KUKA KRL program: MyProgram_079().src

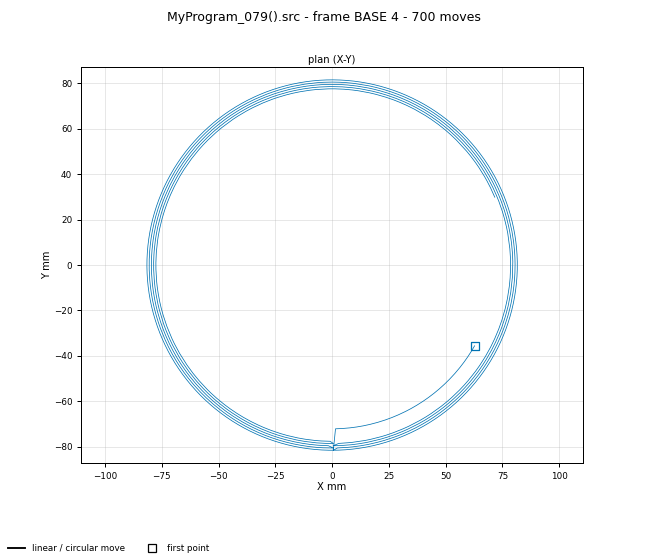
[picture p0: tool path of MyProgram_079().src in frame BASE 4, 700 of 700 moves have a stored position in this frame; points joined in program order, loops and branches not executed]
&ACCESS RVP
&REL 1
&PARAM TEMPLATE = C:\KRC\Roboter\Template\vorgabe
&PARAM EDITMASK = *
DEF MyProgram_079()
; ---- Setting reference (Base) ----
$BASE = BASE_DATA[4]

; --------------------------
; ---- Setting tool (TCP) ----
$TOOL = TOOL_DATA[3]
; --------------------------

$VEL.CP = VEL_APROX_PRINT
Startdeposition()
$VEL.CP = VEL_PRINT
LIN {X 62.743,Y -35.5612,Z 80,A -35.5056,B 24.9021,C -2.2844,E1 25.1384,E2 119.903} C_DIS
LIN {X 61.3969,Y -37.8376,Z 80,A -37.6345,B 24.9027,C -2.2777,E1 25.1353,E2 122.037} C_DIS
LIN {X 59.7597,Y -40.3719,Z 80,A -39.9948,B 24.9032,C -2.2721,E1 25.1316,E2 124.3987} C_DIS
LIN {X 58.1912,Y -42.6015,Z 80,A -42.2134,B 24.9038,C -2.2647,E1 25.128,E2 126.624} C_DIS
LIN {X 56.2909,Y -45.0843,Z 80,A -44.7326,B 24.9044,C -2.2572,E1 25.1237,E2 129.1493} C_DIS
LIN {X 54.0306,Y -47.7691,Z 80,A -47.4805,B 24.9049,C -2.2512,E1 25.1187,E2 131.8988} C_DIS
LIN {X 51.744,Y -50.2367,Z 80,A -50.1078,B 24.9054,C -2.2459,E1 25.1136,E2 134.5273} C_DIS
LIN {X 49.5214,Y -52.4286,Z 80,A -52.5294,B 24.9057,C -2.2416,E1 25.1087,E2 136.9488} C_DIS
LIN {X 47.2452,Y -54.4891,Z 80,A -54.9859,B 24.9062,C -2.2356,E1 25.1036,E2 139.4099} C_DIS
LIN {X 44.8927,Y -56.4428,Z 80,A -57.3886,B 24.9066,C -2.231,E1 25.0984,E2 141.8143} C_DIS
LIN {X 42.5333,Y -58.2412,Z 80,A -59.7773,B 24.9071,C -2.2252,E1 25.093,E2 144.2081} C_DIS
LIN {X 40.0623,Y -59.9686,Z 80,A -62.2006,B 24.9076,C -2.2197,E1 25.0874,E2 146.6363} C_DIS
LIN {X 37.263,Y -61.7465,Z 80,A -64.7758,B 24.9079,C -2.2164,E1 25.0813,E2 149.2111} C_DIS
LIN {X 34.7417,Y -63.2004,Z 80,A -67.0445,B 24.9081,C -2.2135,E1 25.0758,E2 151.4799} C_DIS
LIN {X 32.4215,Y -64.4207,Z 80,A -69.2156,B 24.9086,C -2.2077,E1 25.0704,E2 153.6588} C_DIS
LIN {X 29.2273,Y -65.9316,Z 80,A -72.0556,B 24.909,C -2.2025,E1 25.0632,E2 156.504} C_DIS
LIN {X 26.2757,Y -67.1618,Z 80,A -74.4953,B 24.909,C -2.2017,E1 25.0569,E2 158.9402} C_DIS
LIN {X 23.4466,Y -68.2022,Z 80,A -76.9337,B 24.9094,C -2.1974,E1 25.0504,E2 161.3837} C_DIS
LIN {X 20.0842,Y -69.2668,Z 80,A -79.7346,B 24.9097,C -2.1942,E1 25.0429,E2 164.1871} C_DIS
LIN {X 16.6714,Y -70.165,Z 80,A -82.321,B 24.9094,C -2.1972,E1 25.036,E2 166.7625} C_DIS
LIN {X 13.7247,Y -70.8008,Z 80,A -84.7485,B 24.9097,C -2.1943,E1 25.0293,E2 169.194} C_DIS
LIN {X 10.8752,Y -71.2942,Z 80,A -87.1416,B 24.91,C -2.1901,E1 25.0227,E2 171.5947} C_DIS
LIN {X 7.9418,Y -71.6799,Z 80,A -89.5264,B 24.9102,C -2.1877,E1 25.0161,E2 173.9832} C_DIS
LIN {X 4.4201,Y -71.9832,Z 80,A -92.175,B 24.91,C -2.1906,E1 25.0087,E2 176.6238} C_DIS
LIN {X 1.499,Y -72.1033,Z 80,A -94.5519,B 24.9102,C -2.1884,E1 25.0021,E2 179.0053} C_DIS
LIN {X 1.499,Y -72.1033,Z 80,A -94.5519,B 24.9102,C -2.1884,E1 25.0021,E2 179.0053} C_DIS
Enddeposition()
LIN {X 0.5368,Y -81.5501,Z 81,A -94.2827,B 24.9204,C -2.0597,E1 25.002,E2 179.0416} C_DIS
Startdeposition()
$VEL.CP = VEL_PRINT
LIN {X -1.5341,Y -81.5397,Z 81,A -96.3673,B 24.9219,C -2.0407,E1 24.996,E2 181.1713} C_DIS
LIN {X -4.4685,Y -81.4316,Z 81,A -98.4471,B 24.9219,C -2.04,E1 24.9902,E2 183.2532} C_DIS
LIN {X -7.4627,Y -81.212,Z 81,A -100.5636,B 24.9219,C -2.0399,E1 24.9843,E2 185.371} C_DIS
LIN {X -10.4468,Y -80.8822,Z 81,A -102.6737,B 24.9219,C -2.0401,E1 24.9785,E2 187.4818} C_DIS
LIN {X -13.4168,Y -80.4429,Z 81,A -104.7842,B 24.9219,C -2.0407,E1 24.9727,E2 189.593} C_DIS
LIN {X -16.4332,Y -79.8813,Z 81,A -106.9178,B 24.9219,C -2.0421,E1 24.9668,E2 191.7254} C_DIS
LIN {X -19.3623,Y -79.2223,Z 81,A -109.0295,B 24.9217,C -2.0431,E1 24.9611,E2 193.8376} C_DIS
LIN {X -22.2651,Y -78.456,Z 81,A -111.1414,B 24.9217,C -2.0443,E1 24.9554,E2 195.9499} C_DIS
LIN {X -25.075,Y -77.6036,Z 81,A -113.2323,B 24.9216,C -2.045,E1 24.9498,E2 198.0427} C_DIS
LIN {X -27.9764,Y -76.6055,Z 81,A -115.3677,B 24.9214,C -2.0474,E1 24.9442,E2 200.1766} C_DIS
LIN {X -30.716,Y -75.5487,Z 81,A -117.4594,B 24.9214,C -2.0486,E1 24.9387,E2 202.27} C_DIS
LIN {X -33.4759,Y -74.3669,Z 81,A -119.5737,B 24.9211,C -2.0507,E1 24.9333,E2 204.3844} C_DIS
LIN {X -36.1904,Y -73.0844,Z 81,A -121.6887,B 24.921,C -2.053,E1 24.928,E2 206.4993} C_DIS
LIN {X -38.9139,Y -71.6713,Z 81,A -123.8262,B 24.9207,C -2.0563,E1 24.9227,E2 208.6349} C_DIS
LIN {X -41.4688,Y -70.224,Z 81,A -125.9198,B 24.9206,C -2.0583,E1 24.9177,E2 210.73} C_DIS
LIN {X -44.0254,Y -68.6501,Z 81,A -128.0364,B 24.9203,C -2.0613,E1 24.9127,E2 212.8462} C_DIS
LIN {X -46.5224,Y -66.9831,Z 81,A -130.1279,B 24.92,C -2.0652,E1 24.9078,E2 214.9355} C_DIS
LIN {X -48.9564,Y -65.2254,Z 81,A -132.2705,B 24.9198,C -2.0679,E1 24.903,E2 217.0793} C_DIS
LIN {X -51.3752,Y -63.3377,Z 81,A -134.4108,B 24.9195,C -2.0722,E1 24.8983,E2 219.2173} C_DIS
LIN {X -53.5934,Y -61.4722,Z 81,A -136.4946,B 24.9193,C -2.0747,E1 24.8939,E2 221.303} C_DIS
LIN {X -55.8954,Y -59.3867,Z 81,A -138.6479,B 24.9189,C -2.0799,E1 24.8895,E2 223.4528} C_DIS
LIN {X -58.0434,Y -57.2891,Z 81,A -140.7613,B 24.9185,C -2.0841,E1 24.8853,E2 225.5649} C_DIS
LIN {X -60.0681,Y -55.1624,Z 81,A -142.8642,B 24.9183,C -2.0875,E1 24.8813,E2 227.6689} C_DIS
LIN {X -62.1006,Y -52.8639,Z 81,A -145.0065,B 24.9179,C -2.0928,E1 24.8774,E2 229.8084} C_DIS
LIN {X -64.0043,Y -50.5423,Z 81,A -147.127,B 24.9175,C -2.0974,E1 24.8736,E2 231.9278} C_DIS
LIN {X -65.8212,Y -48.1523,Z 81,A -149.2477,B 24.9171,C -2.1022,E1 24.8701,E2 234.0473} C_DIS
LIN {X -67.512,Y -45.7516,Z 81,A -151.3463,B 24.9168,C -2.1064,E1 24.8668,E2 236.1462} C_DIS
LIN {X -69.1852,Y -43.1797,Z 81,A -153.4902,B 24.9163,C -2.1122,E1 24.8635,E2 238.287} C_DIS
LIN {X -70.6947,Y -40.6611,Z 81,A -155.5896,B 24.916,C -2.1167,E1 24.8606,E2 240.3866} C_DIS
LIN {X -72.1435,Y -38.0315,Z 81,A -157.7117,B 24.9155,C -2.122,E1 24.8577,E2 242.5072} C_DIS
LIN {X -73.523,Y -35.2909,Z 81,A -159.8565,B 24.915,C -2.1283,E1 24.8551,E2 244.6487} C_DIS
LIN {X -74.7458,Y -32.6212,Z 81,A -161.9566,B 24.9147,C -2.1331,E1 24.8527,E2 246.7488} C_DIS
LIN {X -75.8703,Y -29.9127,Z 81,A -164.0576,B 24.9143,C -2.1379,E1 24.8505,E2 248.85} C_DIS
LIN {X -76.9648,Y -26.972,Z 81,A -166.2057,B 24.9136,C -2.1458,E1 24.8485,E2 250.9914} C_DIS
LIN {X -77.8859,Y -24.1838,Z 81,A -168.3262,B 24.9133,C -2.1505,E1 24.8466,E2 253.113} C_DIS
LIN {X -78.7405,Y -21.237,Z 81,A -170.4721,B 24.9127,C -2.1572,E1 24.845,E2 255.2552} C_DIS
LIN {X -79.4688,Y -18.3244,Z 81,A -172.5959,B 24.9122,C -2.1632,E1 24.8436,E2 257.377} C_DIS
LIN {X -80.0894,Y -15.3869,Z 81,A -174.7195,B 24.9117,C -2.1693,E1 24.8424,E2 259.4986} C_DIS
LIN {X -80.6015,Y -12.4286,Z 81,A -176.8435,B 24.9112,C -2.1755,E1 24.8415,E2 261.6205} C_DIS
LIN {X -80.9967,Y -9.519,Z 81,A -178.9453,B 24.9108,C -2.181,E1 24.8407,E2 263.7219} C_DIS
LIN {X -81.2974,Y -6.4656,Z 81,A 178.9082,B 24.9102,C -2.188,E1 24.8402,E2 265.8645} C_DIS
LIN {X -81.4775,Y -3.5347,Z 81,A 176.806,B 24.9097,C -2.1935,E1 24.8399,E2 267.9661} C_DIS
LIN {X -81.553,Y -0.483,Z 81,A 174.6524,B 24.9092,C -2.2001,E1 24.8398,E2 270.117} C_DIS
LIN {X -81.5167,Y 2.4687,Z 81,A 172.5572,B 24.9087,C -2.2062,E1 24.8399,E2 272.2103} C_DIS
LIN {X -81.3662,Y 5.5332,Z 81,A 170.4187,B 24.9081,C -2.2135,E1 24.8402,E2 274.3443} C_DIS
LIN {X -81.1074,Y 8.5243,Z 81,A 168.2859,B 24.9076,C -2.2196,E1 24.8408,E2 276.4752} C_DIS
LIN {X -80.7479,Y 11.4386,Z 81,A 166.1841,B 24.9071,C -2.2252,E1 24.8416,E2 278.5763} C_DIS
LIN {X -80.2605,Y 14.4679,Z 81,A 164.0373,B 24.9065,C -2.2322,E1 24.8426,E2 280.7189} C_DIS
LIN {X -79.6736,Y 17.4122,Z 81,A 161.9133,B 24.906,C -2.2385,E1 24.8438,E2 282.8406} C_DIS
LIN {X -78.9787,Y 20.333,Z 81,A 159.7888,B 24.9055,C -2.2447,E1 24.8452,E2 284.9625} C_DIS
LIN {X -78.1956,Y 23.163,Z 81,A 157.6873,B 24.905,C -2.2502,E1 24.8468,E2 287.0633} C_DIS
LIN {X -77.29,Y 26.0255,Z 81,A 155.5633,B 24.9045,C -2.2563,E1 24.8486,E2 289.1848} C_DIS
LIN {X -76.2564,Y 28.9143,Z 81,A 153.4169,B 24.9039,C -2.2631,E1 24.8507,E2 291.3269} C_DIS
LIN {X -75.1404,Y 31.7015,Z 81,A 151.2934,B 24.9034,C -2.2691,E1 24.8529,E2 293.448} C_DIS
LIN {X -73.9505,Y 34.386,Z 81,A 149.1924,B 24.903,C -2.2743,E1 24.8553,E2 295.5481} C_DIS
LIN {X -72.6348,Y 37.0846,Z 81,A 147.0693,B 24.9025,C -2.2801,E1 24.858,E2 297.6687} C_DIS
LIN {X -71.2206,Y 39.7329,Z 81,A 144.9462,B 24.902,C -2.2859,E1 24.8608,E2 299.7893} C_DIS
LIN {X -69.6756,Y 42.3838,Z 81,A 142.801,B 24.9014,C -2.2923,E1 24.8639,E2 301.9304} C_DIS
LIN {X -68.1046,Y 44.8646,Z 81,A 140.7009,B 24.901,C -2.297,E1 24.867,E2 304.0297} C_DIS
LIN {X -66.3689,Y 47.3946,Z 81,A 138.5564,B 24.9005,C -2.3032,E1 24.8705,E2 306.1701} C_DIS
LIN {X -64.6197,Y 49.7531,Z 81,A 136.4568,B 24.9001,C -2.3077,E1 24.874,E2 308.2689} C_DIS
LIN {X -62.8228,Y 52.0037,Z 81,A 134.3726,B 24.8998,C -2.3114,E1 24.8777,E2 310.3541} C_DIS
LIN {X -60.7405,Y 54.4211,Z 81,A 132.1915,B 24.8991,C -2.3186,E1 24.8817,E2 312.5278} C_DIS
LIN {X -58.6963,Y 56.62,Z 81,A 130.0707,B 24.8987,C -2.3235,E1 24.8857,E2 314.6462} C_DIS
LIN {X -56.5725,Y 58.742,Z 81,A 127.9501,B 24.8983,C -2.3282,E1 24.8899,E2 316.7645} C_DIS
LIN {X -54.372,Y 60.7845,Z 81,A 125.8299,B 24.8979,C -2.3327,E1 24.8943,E2 318.8824} C_DIS
LIN {X -52.1486,Y 62.7025,Z 81,A 123.7326,B 24.8976,C -2.3364,E1 24.8988,E2 320.9791} C_DIS
LIN {X -49.8053,Y 64.5794,Z 81,A 121.6131,B 24.8972,C -2.3406,E1 24.9034,E2 323.0965} C_DIS
LIN {X -47.3409,Y 66.4072,Z 81,A 119.4718,B 24.8968,C -2.3453,E1 24.9082,E2 325.2339} C_DIS
LIN {X -44.8646,Y 68.1046,Z 81,A 117.3614,B 24.8964,C -2.3494,E1 24.9131,E2 327.3417} C_DIS
LIN {X -42.3838,Y 69.6756,Z 81,A 115.2575,B 24.8962,C -2.3521,E1 24.9181,E2 329.4458} C_DIS
LIN {X -39.7905,Y 71.1884,Z 81,A 113.1399,B 24.8959,C -2.3556,E1 24.9232,E2 331.5613} C_DIS
LIN {X -37.0846,Y 72.6348,Z 81,A 111.0093,B 24.8955,C -2.3598,E1 24.9285,E2 333.6877} C_DIS
LIN {X -34.386,Y 73.9505,Z 81,A 108.8838,B 24.8953,C -2.3626,E1 24.9338,E2 335.8119} C_DIS
LIN {X -31.7015,Y 75.1404,Z 81,A 106.7899,B 24.8951,C -2.3648,E1 24.9392,E2 337.9057} C_DIS
LIN {X -28.8526,Y 76.2797,Z 81,A 104.652,B 24.8948,C -2.3682,E1 24.9447,E2 340.0401} C_DIS
LIN {X -26.0255,Y 77.29,Z 81,A 102.5368,B 24.8945,C -2.3706,E1 24.9503,E2 342.1536} C_DIS
LIN {X -23.163,Y 78.1956,Z 81,A 100.4222,B 24.8943,C -2.3728,E1 24.956,E2 344.2666} C_DIS
LIN {X -20.333,Y 78.9787,Z 81,A 98.3306,B 24.8943,C -2.3741,E1 24.9616,E2 346.3584} C_DIS
LIN {X -17.4122,Y 79.6736,Z 81,A 96.2169,B 24.8941,C -2.3759,E1 24.9673,E2 348.4706} C_DIS
LIN {X -14.4679,Y 80.2605,Z 81,A 94.1037,B 24.8939,C -2.3774,E1 24.9731,E2 350.5824} C_DIS
LIN {X -11.4386,Y 80.7479,Z 81,A 91.9688,B 24.8938,C -2.3795,E1 24.979,E2 352.7143} C_DIS
LIN {X -8.5243,Y 81.1074,Z 81,A 89.8792,B 24.8938,C -2.3799,E1 24.9848,E2 354.8043} C_DIS
LIN {X -5.5332,Y 81.3662,Z 81,A 87.7676,B 24.8936,C -2.3807,E1 24.9907,E2 356.9147} C_DIS
LIN {X -2.4687,Y 81.5167,Z 81,A 85.6344,B 24.8936,C -2.3821,E1 24.9966,E2 359.0452} C_DIS
LIN {X 0.4674,Y 81.5528,Z 81,A 83.5466,B 24.8936,C -2.3818,E1 25.0025,E2 361.1337} C_DIS
LIN {X 3.5347,Y 81.4775,Z 81,A 81.4145,B 24.8935,C -2.3827,E1 25.0084,E2 363.2631} C_DIS
LIN {X 6.4656,Y 81.2974,Z 81,A 79.3276,B 24.8935,C -2.3819,E1 25.0142,E2 365.3509} C_DIS
LIN {X 9.519,Y 80.9967,Z 81,A 77.1965,B 24.8935,C -2.3823,E1 25.0201,E2 367.4796} C_DIS
LIN {X 12.4938,Y 80.5914,Z 81,A 75.0884,B 24.8935,C -2.3818,E1 25.026,E2 369.5871} C_DIS
LIN {X 15.3869,Y 80.0894,Z 81,A 73.0029,B 24.8937,C -2.3804,E1 25.0317,E2 371.6737} C_DIS
LIN {X 18.3244,Y 79.4688,Z 81,A 70.896,B 24.8937,C -2.3794,E1 25.0374,E2 373.7801} C_DIS
LIN {X 21.237,Y 78.7405,Z 81,A 68.7893,B 24.8939,C -2.3782,E1 25.0431,E2 375.8864} C_DIS
LIN {X 24.1838,Y 77.8859,Z 81,A 66.661,B 24.8939,C -2.3774,E1 25.0488,E2 378.0127} C_DIS
LIN {X 26.972,Y 76.9648,Z 81,A 64.5779,B 24.8941,C -2.3751,E1 25.0543,E2 380.0972} C_DIS
LIN {X 29.8479,Y 75.8958,Z 81,A 62.4507,B 24.8943,C -2.3739,E1 25.0599,E2 382.2227} C_DIS
LIN {X 32.6212,Y 74.7458,Z 81,A 60.347,B 24.8944,C -2.3718,E1 25.0653,E2 384.3264} C_DIS
LIN {X 35.3503,Y 73.4944,Z 81,A 58.2425,B 24.8946,C -2.3695,E1 25.0706,E2 386.431} C_DIS
LIN {X 38.0315,Y 72.1435,Z 81,A 56.139,B 24.8949,C -2.367,E1 25.0758,E2 388.5346} C_DIS
LIN {X 40.6611,Y 70.6947,Z 81,A 54.0363,B 24.8951,C -2.3643,E1 25.081,E2 390.6376} C_DIS
LIN {X 43.1797,Y 69.1852,Z 81,A 51.9561,B 24.8954,C -2.3607,E1 25.0859,E2 392.7198} C_DIS
LIN {X 45.7516,Y 67.512,Z 81,A 49.8319,B 24.8956,C -2.3582,E1 25.0909,E2 394.8428} C_DIS
LIN {X 48.2055,Y 65.7822,Z 81,A 47.7307,B 24.8959,C -2.3549,E1 25.0956,E2 396.9445} C_DIS
LIN {X 50.5941,Y 63.9634,Z 81,A 45.6295,B 24.8963,C -2.3514,E1 25.1003,E2 399.0464} C_DIS
LIN {X 52.8639,Y 62.1006,Z 81,A 43.551,B 24.8966,C -2.347,E1 25.1047,E2 401.1272} C_DIS
LIN {X 55.1138,Y 60.1127,Z 81,A 41.4509,B 24.897,C -2.3431,E1 25.1091,E2 403.2281} C_DIS
LIN {X 57.2891,Y 58.0434,Z 81,A 39.3512,B 24.8973,C -2.339,E1 25.1133,E2 405.3287} C_DIS
LIN {X 59.3867,Y 55.8954,Z 81,A 37.2519,B 24.8977,C -2.3348,E1 25.1174,E2 407.4289} C_DIS
LIN {X 61.4472,Y 53.622,Z 81,A 35.1661,B 24.898,C -2.3321,E1 25.1213,E2 409.5117} C_DIS
LIN {X 63.3377,Y 51.3752,Z 81,A 33.0545,B 24.8985,C -2.3258,E1 25.125,E2 411.6285} C_DIS
LIN {X 65.1857,Y 49.0091,Z 81,A 30.9562,B 24.8989,C -2.3211,E1 25.1286,E2 413.728} C_DIS
LIN {X 66.9585,Y 46.5578,Z 81,A 28.8509,B 24.8993,C -2.3165,E1 25.132,E2 415.8341} C_DIS
LIN {X 68.6144,Y 44.081,Z 81,A 26.7609,B 24.8998,C -2.3112,E1 25.1352,E2 417.926} C_DIS
LIN {X 70.1905,Y 41.5256,Z 81,A 24.6638,B 24.9002,C -2.3061,E1 25.1383,E2 420.0245} C_DIS
LIN {X 71.7028,Y 38.8559,Z 81,A 22.5447,B 24.9006,C -2.3015,E1 25.1411,E2 422.1435} C_DIS
LIN {X 73.0551,Y 36.2495,Z 81,A 20.4705,B 24.9011,C -2.2954,E1 25.1438,E2 424.221} C_DIS
LIN {X 74.3398,Y 33.536,Z 81,A 18.374,B 24.9016,C -2.2899,E1 25.1462,E2 426.3191} C_DIS
LIN {X 75.5487,Y 30.716,Z 81,A 16.2558,B 24.902,C -2.285,E1 25.1485,E2 428.4373} C_DIS
LIN {X 76.6281,Y 27.9144,Z 81,A 14.16,B 24.9025,C -2.2793,E1 25.1506,E2 430.535} C_DIS
LIN {X 77.5833,Y 25.1378,Z 81,A 12.0866,B 24.9031,C -2.2728,E1 25.1524,E2 432.6119} C_DIS
LIN {X 78.456,Y 22.2651,Z 81,A 9.9911,B 24.9036,C -2.2669,E1 25.1541,E2 434.7093} C_DIS
LIN {X 79.2379,Y 19.2982,Z 81,A 7.8736,B 24.904,C -2.2616,E1 25.1555,E2 436.8272} C_DIS
LIN {X 79.8813,Y 16.4332,Z 81,A 5.8008,B 24.9046,C -2.255,E1 25.1568,E2 438.9036} C_DIS
LIN {X 80.4429,Y 13.4168,Z 81,A 3.6837,B 24.9051,C -2.2495,E1 25.1578,E2 441.0211} C_DIS
LIN {X 80.8822,Y 10.4468,Z 81,A 1.5889,B 24.9056,C -2.2434,E1 25.1586,E2 443.1181} C_DIS
LIN {X 81.212,Y 7.4627,Z 81,A -0.506,B 24.9061,C -2.2372,E1 25.1592,E2 445.2151} C_DIS
LIN {X 81.4316,Y 4.4685,Z 81,A -2.6004,B 24.9066,C -2.231,E1 25.1596,E2 447.3118} C_DIS
LIN {X 81.5397,Y 1.5341,Z 81,A -4.6754,B 24.9072,C -2.2241,E1 25.1598,E2 449.3908} C_DIS
LIN {X 81.5311,Y -2.0015,Z 81,A -7.2342,B 24.9081,C -2.2137,E1 25.1597,E2 451.9589} C_DIS
LIN {X 81.4022,Y -5.0011,Z 81,A -9.321,B 24.9086,C -2.2077,E1 25.1594,E2 454.0475} C_DIS
LIN {X 81.1736,Y -7.8785,Z 81,A -11.3675,B 24.9092,C -2.2006,E1 25.1589,E2 456.0985} C_DIS
LIN {X 80.8137,Y -10.9758,Z 81,A -13.51,B 24.9096,C -2.1952,E1 25.1581,E2 458.2412} C_DIS
LIN {X 80.355,Y -13.9429,Z 81,A -15.6046,B 24.9101,C -2.1889,E1 25.1572,E2 460.3382} C_DIS
LIN {X 79.7873,Y -16.8911,Z 81,A -17.699,B 24.9106,C -2.1827,E1 25.156,E2 462.435} C_DIS
LIN {X 79.1115,Y -19.8164,Z 81,A -19.7938,B 24.9111,C -2.1766,E1 25.1546,E2 464.5323} C_DIS
LIN {X 78.3285,Y -22.7149,Z 81,A -21.9076,B 24.9117,C -2.1698,E1 25.153,E2 466.6499} C_DIS
LIN {X 77.4394,Y -25.5825,Z 81,A -23.9836,B 24.9121,C -2.1643,E1 25.1513,E2 468.7271} C_DIS
LIN {X 76.4453,Y -28.4155,Z 81,A -26.0978,B 24.9127,C -2.1577,E1 25.1492,E2 470.8451} C_DIS
LIN {X 75.3476,Y -31.21,Z 81,A -28.1931,B 24.9132,C -2.1517,E1 25.1471,E2 472.9429} C_DIS
LIN {X 74.1478,Y -33.9622,Z 81,A -30.2692,B 24.9136,C -2.1465,E1 25.1447,E2 475.0202} C_DIS
LIN {X 72.8475,Y -36.6683,Z 81,A -32.384,B 24.9141,C -2.1401,E1 25.1421,E2 477.1388} C_DIS
LIN {X 71.4485,Y -39.3248,Z 81,A -34.4799,B 24.9146,C -2.1343,E1 25.1393,E2 479.2371} C_DIS
LIN {X 69.9526,Y -41.928,Z 81,A -36.5568,B 24.915,C -2.1293,E1 25.1363,E2 481.3152} C_DIS
LIN {X 68.362,Y -44.4743,Z 81,A -38.6723,B 24.9155,C -2.1232,E1 25.1332,E2 483.4345} C_DIS
LIN {X 66.6787,Y -46.9604,Z 81,A -40.7495,B 24.9158,C -2.1184,E1 25.1299,E2 485.5128} C_DIS
LIN {X 64.905,Y -49.3828,Z 81,A -42.8464,B 24.9163,C -2.1132,E1 25.1263,E2 487.6121} C_DIS
LIN {X 63.0859,Y -51.6858,Z 81,A -44.9027,B 24.9167,C -2.1079,E1 25.1227,E2 489.6712} C_DIS
LIN {X 61.0963,Y -54.0237,Z 81,A -47.0602,B 24.9171,C -2.1024,E1 25.1188,E2 491.8321} C_DIS
LIN {X 59.0664,Y -56.2359,Z 81,A -49.1388,B 24.9174,C -2.0981,E1 25.1148,E2 493.9116} C_DIS
LIN {X 56.9565,Y -58.3719,Z 81,A -51.237,B 24.9178,C -2.0934,E1 25.1107,E2 496.0122} C_DIS
LIN {X 54.7694,Y -60.4287,Z 81,A -53.3546,B 24.9182,C -2.0882,E1 25.1063,E2 498.1335} C_DIS
LIN {X 52.5081,Y -62.4037,Z 81,A -55.4344,B 24.9185,C -2.0844,E1 25.1019,E2 500.2141} C_DIS
LIN {X 50.1756,Y -64.2941,Z 81,A -57.4993,B 24.9188,C -2.0812,E1 25.0974,E2 502.2788} C_DIS
LIN {X 47.7751,Y -66.0974,Z 81,A -59.6525,B 24.9192,C -2.0755,E1 25.0925,E2 504.438} C_DIS
LIN {X 45.3099,Y -67.811,Z 81,A -61.7527,B 24.9195,C -2.0716,E1 25.0877,E2 506.5402} C_DIS
LIN {X 42.7832,Y -69.4328,Z 81,A -63.8534,B 24.9198,C -2.0679,E1 25.0827,E2 508.643} C_DIS
LIN {X 40.1986,Y -70.9605,Z 81,A -65.9353,B 24.92,C -2.0649,E1 25.0777,E2 510.7256} C_DIS
LIN {X 37.5595,Y -72.392,Z 81,A -68.0556,B 24.9203,C -2.061,E1 25.0724,E2 512.8492} C_DIS
LIN {X 34.8695,Y -73.7254,Z 81,A -70.1577,B 24.9206,C -2.0579,E1 25.0671,E2 514.9532} C_DIS
LIN {X 32.1323,Y -74.9589,Z 81,A -72.2601,B 24.9208,C -2.055,E1 25.0617,E2 517.0574} C_DIS
LIN {X 29.3515,Y -76.0908,Z 81,A -74.3439,B 24.921,C -2.0528,E1 25.0563,E2 519.1416} C_DIS
LIN {X 26.5309,Y -77.1196,Z 81,A -76.4662,B 24.9212,C -2.0497,E1 25.0507,E2 521.267} C_DIS
LIN {X 23.6744,Y -78.0439,Z 81,A -78.5513,B 24.9214,C -2.048,E1 25.0452,E2 523.3524} C_DIS
LIN {X 20.7857,Y -78.8624,Z 81,A -80.6554,B 24.9215,C -2.0459,E1 25.0395,E2 525.4581} C_DIS
LIN {X 17.8689,Y -79.574,Z 81,A -82.7603,B 24.9217,C -2.044,E1 25.0338,E2 527.5644} C_DIS
LIN {X 14.9279,Y -80.1778,Z 81,A -84.8851,B 24.9218,C -2.0418,E1 25.0279,E2 529.692} C_DIS
LIN {X 11.9667,Y -80.6729,Z 81,A -86.9911,B 24.9219,C -2.0404,E1 25.0221,E2 531.7993} C_DIS
LIN {X 8.9892,Y -81.0587,Z 81,A -89.0976,B 24.922,C -2.0392,E1 25.0163,E2 533.9071} C_DIS
LIN {X 5.9996,Y -81.3347,Z 81,A -91.2046,B 24.9221,C -2.0382,E1 25.0104,E2 536.0153} C_DIS
LIN {X 3.0018,Y -81.5004,Z 81,A -93.2931,B 24.9221,C -2.038,E1 25.0046,E2 538.1036} C_DIS
LIN {X 0.5368,Y -81.5501,Z 81,A -94.2824,B 24.9205,C -2.0596,E1 25.002,E2 539.0414} C_DIS
Enddeposition()
LIN {X 0.5368,Y -81.5501,Z 81,A -94.2824,B 24.9205,C -2.0596,E1 25.002,E2 539.0414} C_DIS
Startdeposition()
$VEL.CP = VEL_PRINT
LIN {X 2.3737,Y -80.5326,Z 81,A -92.7908,B 24.9187,C -2.0825,E1 25.0063,E2 537.4957} C_DIS
LIN {X 6.7156,Y -80.2877,Z 81,A -89.5811,B 24.9183,C -2.0874,E1 25.0153,E2 534.276} C_DIS
LIN {X 9.0628,Y -80.0568,Z 81,A -87.3356,B 24.9169,C -2.1055,E1 25.0216,E2 531.9892} C_DIS
LIN {X 12.3593,Y -79.6139,Z 81,A -85.5383,B 24.9181,C -2.0899,E1 25.0265,E2 530.2303} C_DIS
LIN {X 15.7366,Y -79.0172,Z 81,A -83.0361,B 24.9178,C -2.0938,E1 25.0334,E2 527.7218} C_DIS
LIN {X 20.0644,Y -78.0291,Z 81,A -80.0615,B 24.918,C -2.0913,E1 25.0414,E2 524.7573} C_DIS
LIN {X 23.1372,Y -77.1742,Z 81,A -77.832,B 24.9179,C -2.0927,E1 25.0474,E2 522.5285} C_DIS
LIN {X 27.5884,Y -75.6968,Z 81,A -74.4245,B 24.9174,C -2.099,E1 25.0564,E2 519.1126} C_DIS
LIN {X 30.5902,Y -74.5347,Z 81,A -72.1179,B 24.9171,C -2.1027,E1 25.0624,E2 516.8025} C_DIS
LIN {X 33.5873,Y -73.234,Z 81,A -69.7673,B 24.9167,C -2.1071,E1 25.0684,E2 514.4474} C_DIS
LIN {X 36.569,Y -71.7903,Z 81,A -67.4679,B 24.9166,C -2.1092,E1 25.0742,E2 512.1492} C_DIS
LIN {X 39.4625,Y -70.2416,Z 81,A -65.0553,B 24.9161,C -2.1156,E1 25.0801,E2 509.7283} C_DIS
LIN {X 42.2836,Y -68.5817,Z 81,A -62.7419,B 24.9158,C -2.1195,E1 25.0856,E2 507.413} C_DIS
LIN {X 45.0321,Y -66.8076,Z 81,A -60.499,B 24.9156,C -2.1214,E1 25.0908,E2 505.173} C_DIS
LIN {X 47.767,Y -64.8806,Z 81,A -58.0571,B 24.9151,C -2.1282,E1 25.0964,E2 502.7234} C_DIS
LIN {X 50.4956,Y -62.7807,Z 81,A -55.6497,B 24.9147,C -2.1322,E1 25.1017,E2 500.3156} C_DIS
LIN {X 53.1214,Y -60.5745,Z 81,A -53.1992,B 24.9143,C -2.1381,E1 25.1069,E2 497.8608} C_DIS
LIN {X 55.5812,Y -58.3272,Z 81,A -50.8454,B 24.9139,C -2.1431,E1 25.1117,E2 495.5048} C_DIS
LIN {X 57.9436,Y -55.9792,Z 81,A -48.5126,B 24.9135,C -2.1477,E1 25.1162,E2 493.171} C_DIS
LIN {X 59.9721,Y -53.8004,Z 81,A -46.3803,B 24.913,C -2.1535,E1 25.1203,E2 491.0344} C_DIS
LIN {X 62.2149,Y -51.1916,Z 81,A -43.932,B 24.9125,C -2.1599,E1 25.1247,E2 488.5822} C_DIS
LIN {X 64.3316,Y -48.5035,Z 81,A -41.5852,B 24.9122,C -2.1636,E1 25.1287,E2 486.2377} C_DIS
LIN {X 66.2625,Y -45.8306,Z 81,A -39.225,B 24.9116,C -2.1705,E1 25.1325,E2 483.8728} C_DIS
LIN {X 67.839,Y -43.4626,Z 81,A -37.409,B 24.9117,C -2.1695,E1 25.1352,E2 482.0683} C_DIS
LIN {X 69.6895,Y -40.4303,Z 81,A -34.6946,B 24.9106,C -2.1827,E1 25.1391,E2 479.3365} C_DIS
LIN {X 71.2785,Y -37.5566,Z 81,A -32.4414,B 24.9103,C -2.1869,E1 25.1421,E2 477.0853} C_DIS
LIN {X 72.6952,Y -34.7356,Z 81,A -30.1801,B 24.9097,C -2.1941,E1 25.1449,E2 474.8191} C_DIS
LIN {X 73.9069,Y -32.0767,Z 81,A -28.0065,B 24.9089,C -2.2034,E1 25.1474,E2 472.6353} C_DIS
LIN {X 75.2146,Y -28.8796,Z 81,A -25.7389,B 24.9089,C -2.2047,E1 25.1497,E2 470.3771} C_DIS
LIN {X 76.1166,Y -26.4096,Z 81,A -23.3881,B 24.907,C -2.2262,E1 25.1519,E2 467.9889} C_DIS
LIN {X 77.4487,Y -22.2008,Z 81,A -20.6607,B 24.9073,C -2.2225,E1 25.1541,E2 465.2857} C_DIS
LIN {X 78.3258,Y -18.8743,Z 81,A -18.2324,B 24.9067,C -2.2296,E1 25.1557,E2 462.8547} C_DIS
LIN {X 78.8255,Y -16.6701,Z 81,A -16.2471,B 24.9053,C -2.247,E1 25.1569,E2 460.8399} C_DIS
LIN {X 79.6176,Y -12.3358,Z 81,A -13.9574,B 24.9068,C -2.2295,E1 25.158,E2 458.6049} C_DIS
LIN {X 80.0508,Y -9.1139,Z 81,A -11.2642,B 24.9051,C -2.2492,E1 25.1589,E2 455.881} C_DIS
LIN {X 80.3421,Y -6.0346,Z 81,A -9.0617,B 24.9045,C -2.2563,E1 25.1595,E2 453.6748} C_DIS
LIN {X 80.5015,Y -3.2671,Z 81,A -7.0297,B 24.9038,C -2.2646,E1 25.1597,E2 451.6353} C_DIS
LIN {X 80.5677,Y 0.2486,Z 81,A -4.6645,B 24.9035,C -2.2682,E1 25.1597,E2 449.2758} C_DIS
LIN {X 80.5049,Y 3.188,Z 81,A -2.5943,B 24.903,C -2.2742,E1 25.1596,E2 447.2038} C_DIS
LIN {X 80.3371,Y 6.0978,Z 81,A -0.2536,B 24.9017,C -2.2894,E1 25.1591,E2 444.8409} C_DIS
LIN {X 79.9461,Y 9.9936,Z 81,A 3.4087,B 24.8984,C -2.327,E1 25.1579,E2 441.1117} C_DIS
LIN {X 79.1646,Y 14.9721,Z 81,A 5.659,B 24.9012,C -2.2945,E1 25.1568,E2 438.9513} C_DIS
LIN {X 77.7971,Y 20.9462,Z 81,A 10.1729,B 24.8996,C -2.3127,E1 25.1539,E2 434.4204} C_DIS
LIN {X 76.8637,Y 24.1494,Z 81,A 12.6212,B 24.8988,C -2.3223,E1 25.1519,E2 431.9636} C_DIS
LIN {X 75.7107,Y 27.5504,Z 81,A 15.0618,B 24.8985,C -2.3261,E1 25.1496,E2 429.5276} C_DIS
LIN {X 74.659,Y 30.2849,Z 81,A 17.1278,B 24.898,C -2.3316,E1 25.1475,E2 427.4601} C_DIS
LIN {X 73.1933,Y 33.6747,Z 81,A 19.7392,B 24.8974,C -2.3385,E1 25.1445,E2 424.8466} C_DIS
LIN {X 71.8343,Y 36.4828,Z 81,A 21.8781,B 24.8971,C -2.3421,E1 25.1419,E2 422.7106} C_DIS
LIN {X 70.2193,Y 39.5023,Z 81,A 24.3755,B 24.8963,C -2.3506,E1 25.1385,E2 420.2061} C_DIS
LIN {X 68.5467,Y 42.3396,Z 81,A 26.7423,B 24.8957,C -2.3575,E1 25.1351,E2 417.8351} C_DIS
LIN {X 66.7041,Y 45.1851,Z 81,A 28.9449,B 24.8957,C -2.3571,E1 25.1317,E2 415.6445} C_DIS
LIN {X 64.7297,Y 47.9729,Z 81,A 31.5875,B 24.8946,C -2.3698,E1 25.1274,E2 412.9847} C_DIS
LIN {X 62.4637,Y 50.8867,Z 81,A 34.1374,B 24.8943,C -2.3736,E1 25.1229,E2 410.4376} C_DIS
LIN {X 59.209,Y 54.6395,Z 81,A 37.6024,B 24.8938,C -2.3794,E1 25.1165,E2 406.9744} C_DIS
LIN {X 57.0379,Y 56.9031,Z 81,A 39.8671,B 24.8932,C -2.3852,E1 25.1121,E2 404.7056} C_DIS
LIN {X 54.9645,Y 58.9078,Z 81,A 41.9663,B 24.8927,C -2.3909,E1 25.1078,E2 402.6016} C_DIS
LIN {X 52.3298,Y 61.2595,Z 81,A 44.422,B 24.8924,C -2.3941,E1 25.1027,E2 400.1481} C_DIS
LIN {X 50.6302,Y 62.6715,Z 81,A 46.4336,B 24.8909,C -2.4107,E1 25.0982,E2 398.1049} C_DIS
LIN {X 47.5653,Y 65.0282,Z 81,A 48.6853,B 24.8919,C -2.4,E1 25.0933,E2 395.8864} C_DIS
LIN {X 44.9476,Y 66.8648,Z 81,A 50.984,B 24.8915,C -2.4045,E1 25.088,E2 393.585} C_DIS
LIN {X 42.2198,Y 68.6207,Z 81,A 53.3044,B 24.8911,C -2.4084,E1 25.0825,E2 391.2627} C_DIS
LIN {X 40.0642,Y 69.8999,Z 81,A 55.1,B 24.8909,C -2.4114,E1 25.0781,E2 389.4655} C_DIS
LIN {X 37.6818,Y 71.2126,Z 81,A 57.0524,B 24.8906,C -2.4145,E1 25.0733,E2 387.5113} C_DIS
LIN {X 34.4865,Y 72.8149,Z 81,A 59.3682,B 24.8909,C -2.4107,E1 25.0675,E2 385.2106} C_DIS
LIN {X 31.9777,Y 73.95,Z 81,A 61.4746,B 24.8903,C -2.4174,E1 25.0621,E2 383.0936} C_DIS
LIN {X 28.9795,Y 75.1767,Z 81,A 63.8035,B 24.8901,C -2.4204,E1 25.0561,E2 380.7628} C_DIS
LIN {X 25.9351,Y 76.2793,Z 81,A 66.0103,B 24.8901,C -2.4195,E1 25.0503,E2 378.5624} C_DIS
LIN {X 22.8488,Y 77.2597,Z 81,A 68.3905,B 24.8898,C -2.4235,E1 25.0439,E2 376.177} C_DIS
LIN {X 19.5226,Y 78.1677,Z 81,A 70.8635,B 24.8896,C -2.4257,E1 25.0372,E2 373.7028} C_DIS
LIN {X 16.0828,Y 78.9461,Z 81,A 73.439,B 24.8893,C -2.4288,E1 25.0302,E2 371.123} C_DIS
LIN {X 9.5594,Y 79.9986,Z 81,A 77.8609,B 24.8899,C -2.422,E1 25.018,E2 366.7215} C_DIS
LIN {X 6.2156,Y 80.3277,Z 81,A 80.44,B 24.8894,C -2.4277,E1 25.0108,E2 364.1303} C_DIS
LIN {X 3.3358,Y 80.4985,Z 81,A 83.004,B 24.888,C -2.4425,E1 25.0036,E2 361.532} C_DIS
LIN {X 0.0164,Y 80.5686,Z 81,A 84.7626,B 24.8897,C -2.4246,E1 24.9988,E2 359.8159} C_DIS
LIN {X -3.8251,Y 80.4775,Z 81,A 87.7572,B 24.8891,C -2.4313,E1 24.9904,E2 356.8049} C_DIS
LIN {X -6.4775,Y 80.3067,Z 81,A 89.8326,B 24.8887,C -2.4358,E1 24.9846,E2 354.7181} C_DIS
LIN {X -12.0438,Y 79.6627,Z 81,A 93.9174,B 24.8887,C -2.4361,E1 24.9733,E2 350.6293} C_DIS
LIN {X -17.6377,Y 78.6143,Z 81,A 97.2506,B 24.8908,C -2.4127,E1 24.9643,E2 347.348} C_DIS
LIN {X -20.1158,Y 78.0159,Z 81,A 99.3155,B 24.8903,C -2.418,E1 24.9586,E2 345.2675} C_DIS
LIN {X -23.3267,Y 77.1179,Z 81,A 101.7242,B 24.8904,C -2.4165,E1 24.9522,E2 342.8586} C_DIS
LIN {X -26.4247,Y 76.1113,Z 81,A 103.6815,B 24.8916,C -2.4038,E1 24.9471,E2 340.9277} C_DIS
LIN {X -28.5901,Y 75.3242,Z 81,A 106.0592,B 24.8899,C -2.4221,E1 24.9407,E2 338.5016} C_DIS
LIN {X -34.0629,Y 73.0127,Z 81,A 109.8055,B 24.8917,C -2.4027,E1 24.9312,E2 334.7925} C_DIS
LIN {X -37.2985,Y 71.4145,Z 81,A 112.4681,B 24.8917,C -2.4012,E1 24.9246,E2 332.1264} C_DIS
LIN {X -40.2552,Y 69.7901,Z 81,A 114.908,B 24.8921,C -2.3982,E1 24.9187,E2 329.6865} C_DIS
LIN {X -43.1458,Y 68.0423,Z 81,A 117.3287,B 24.8924,C -2.3942,E1 24.9129,E2 327.2677} C_DIS
LIN {X -45.9035,Y 66.2118,Z 81,A 119.6216,B 24.893,C -2.388,E1 24.9076,E2 324.9819} C_DIS
LIN {X -48.4343,Y 64.3836,Z 81,A 121.8432,B 24.8934,C -2.3835,E1 24.9027,E2 322.7632} C_DIS
LIN {X -50.9037,Y 62.4499,Z 81,A 124.0937,B 24.8938,C -2.3793,E1 24.8978,E2 320.5145} C_DIS
LIN {X -53.2413,Y 60.4698,Z 81,A 126.3008,B 24.8941,C -2.3752,E1 24.8931,E2 318.3085} C_DIS
LIN {X -55.5834,Y 58.3248,Z 81,A 128.6906,B 24.8943,C -2.3734,E1 24.8882,E2 315.9131} C_DIS
LIN {X -58.1179,Y 55.7984,Z 81,A 131.0735,B 24.8952,C -2.363,E1 24.8836,E2 313.5448} C_DIS
LIN {X -60.1539,Y 53.5973,Z 81,A 133.2379,B 24.8956,C -2.3585,E1 24.8795,E2 311.3814} C_DIS
LIN {X -61.8965,Y 51.5748,Z 81,A 135.1031,B 24.8961,C -2.3528,E1 24.8762,E2 309.5213} C_DIS
LIN {X -64.2116,Y 48.6632,Z 81,A 137.8528,B 24.8965,C -2.3486,E1 24.8714,E2 306.7688} C_DIS
LIN {X -66.0547,Y 46.1295,Z 81,A 140.0335,B 24.8971,C -2.3413,E1 24.8679,E2 304.5948} C_DIS
LIN {X -67.715,Y 43.6559,Z 81,A 142.1662,B 24.8976,C -2.3358,E1 24.8646,E2 302.4644} C_DIS
LIN {X -69.3556,Y 40.9991,Z 81,A 144.446,B 24.898,C -2.3311,E1 24.8614,E2 300.1842} C_DIS
LIN {X -71.7233,Y 36.7001,Z 81,A 147.8626,B 24.8991,C -2.3191,E1 24.8569,E2 296.7782} C_DIS
LIN {X -73.2979,Y 33.4467,Z 81,A 150.5641,B 24.8995,C -2.3148,E1 24.8536,E2 294.0722} C_DIS
LIN {X -74.5367,Y 30.5853,Z 81,A 152.7602,B 24.9001,C -2.3076,E1 24.8512,E2 291.8811} C_DIS
LIN {X -75.7008,Y 27.5773,Z 81,A 155.0088,B 24.9008,C -2.2994,E1 24.849,E2 289.6394} C_DIS
LIN {X -76.6797,Y 24.7257,Z 81,A 157.206,B 24.9013,C -2.2942,E1 24.8471,E2 287.4421} C_DIS
LIN {X -77.5849,Y 21.7203,Z 81,A 159.5892,B 24.9015,C -2.2912,E1 24.8452,E2 285.0524} C_DIS
LIN {X -78.4153,Y 18.5015,Z 81,A 161.9096,B 24.9022,C -2.2826,E1 24.8437,E2 282.7388} C_DIS
LIN {X -79.1147,Y 15.2313,Z 81,A 164.3339,B 24.9028,C -2.2763,E1 24.8424,E2 280.3154} C_DIS
LIN {X -79.6799,Y 11.9328,Z 81,A 166.7196,B 24.9034,C -2.2689,E1 24.8413,E2 277.9332} C_DIS
LIN {X -80.1111,Y 8.5655,Z 81,A 169.2263,B 24.9039,C -2.2636,E1 24.8405,E2 275.4241} C_DIS
LIN {X -80.3271,Y 6.2226,Z 81,A 171.5343,B 24.9029,C -2.2747,E1 24.84,E2 273.0756} C_DIS
LIN {X -80.5308,Y 2.4337,Z 81,A 173.1671,B 24.906,C -2.2386,E1 24.8399,E2 271.5194} C_DIS
LIN {X -80.5457,Y -1.9141,Z 81,A 176.4255,B 24.9065,C -2.2329,E1 24.8399,E2 268.2547} C_DIS
LIN {X -80.2966,Y -6.6042,Z 81,A 179.8384,B 24.9072,C -2.2242,E1 24.8404,E2 264.8421} C_DIS
LIN {X -79.9955,Y -9.5864,Z 81,A -177.8184,B 24.9073,C -2.223,E1 24.8411,E2 262.4879} C_DIS
LIN {X -79.5897,Y -12.5157,Z 81,A -175.7665,B 24.908,C -2.2151,E1 24.842,E2 260.4425} C_DIS
LIN {X -79.0283,Y -15.6799,Z 81,A -173.3684,B 24.9083,C -2.211,E1 24.8432,E2 258.0401} C_DIS
LIN {X -78.2987,Y -18.9855,Z 81,A -171.0486,B 24.9091,C -2.2014,E1 24.8447,E2 255.7296} C_DIS
LIN {X -77.4427,Y -22.2221,Z 81,A -168.6082,B 24.9096,C -2.1957,E1 24.8465,E2 253.2884} C_DIS
LIN {X -76.5217,Y -25.2139,Z 81,A -166.3704,B 24.9101,C -2.1894,E1 24.8484,E2 251.053} C_DIS
LIN {X -75.5306,Y -28.0441,Z 81,A -164.2207,B 24.9106,C -2.1837,E1 24.8504,E2 248.9049} C_DIS
LIN {X -73.5052,Y -32.9868,Z 81,A -160.4507,B 24.9115,C -2.1721,E1 24.8545,E2 245.1416} C_DIS
LIN {X -72.0647,Y -36.0261,Z 81,A -158.0187,B 24.912,C -2.1665,E1 24.8575,E2 242.7097} C_DIS
LIN {X -70.5822,Y -38.8518,Z 81,A -155.676,B 24.9123,C -2.1623,E1 24.8606,E2 240.3646} C_DIS
LIN {X -68.8797,Y -41.7938,Z 81,A -153.3682,B 24.9131,C -2.1531,E1 24.8639,E2 238.0669} C_DIS
LIN {X -67.2835,Y -44.3177,Z 81,A -151.2336,B 24.9135,C -2.1479,E1 24.8671,E2 235.9338} C_DIS
LIN {X -65.2891,Y -47.209,Z 81,A -148.5948,B 24.9137,C -2.1455,E1 24.8713,E2 233.2879} C_DIS
LIN {X -63.3053,Y -49.8356,Z 81,A -146.4676,B 24.9146,C -2.1342,E1 24.8749,E2 231.1774} C_DIS
LIN {X -60.778,Y -52.8884,Z 81,A -142.9401,B 24.9136,C -2.1469,E1 24.8814,E2 227.6036} C_DIS
LIN {X -58.008,Y -55.9124,Z 81,A -140.4413,B 24.915,C -2.1292,E1 24.8861,E2 225.1361} C_DIS
LIN {X -55.4335,Y -58.4668,Z 81,A -137.9164,B 24.9155,C -2.1225,E1 24.8912,E2 222.6168} C_DIS
LIN {X -52.6141,Y -61.0173,Z 81,A -134.7467,B 24.9149,C -2.13,E1 24.8979,E2 219.4166} C_DIS
LIN {X -48.9059,Y -64.027,Z 81,A -131.7962,B 24.9164,C -2.1116,E1 24.9043,E2 216.499} C_DIS
LIN {X -46.4037,Y -65.8639,Z 81,A -129.5585,B 24.9166,C -2.1087,E1 24.9094,E2 214.2604} C_DIS
LIN {X -43.8306,Y -67.6028,Z 81,A -127.6616,B 24.9176,C -2.0967,E1 24.9137,E2 212.3859} C_DIS
LIN {X -41.4618,Y -69.0814,Z 81,A -125.4334,B 24.9173,C -2.1004,E1 24.9191,E2 210.1418} C_DIS
LIN {X -38.3636,Y -70.8475,Z 81,A -122.8467,B 24.9174,C -2.0984,E1 24.9254,E2 207.5524} C_DIS
LIN {X -35.4358,Y -72.3573,Z 81,A -120.4529,B 24.9175,C -2.097,E1 24.9314,E2 205.1557} C_DIS
LIN {X -32.521,Y -73.7132,Z 81,A -118.1846,B 24.9178,C -2.094,E1 24.9371,E2 202.8891} C_DIS
LIN {X -29.5668,Y -74.9463,Z 81,A -115.8343,B 24.9178,C -2.0938,E1 24.9432,E2 200.5338} C_DIS
LIN {X -26.5662,Y -76.0617,Z 81,A -113.5888,B 24.918,C -2.091,E1 24.9491,E2 198.2906} C_DIS
LIN {X -23.2711,Y -77.1344,Z 81,A -111.2416,B 24.9184,C -2.0858,E1 24.9554,E2 195.9516} C_DIS
LIN {X -20.3864,Y -77.9464,Z 81,A -109.0614,B 24.9184,C -2.0859,E1 24.9613,E2 193.7679} C_DIS
LIN {X -17.0688,Y -78.7387,Z 81,A -106.0317,B 24.9171,C -2.1023,E1 24.9696,E2 190.6953} C_DIS
LIN {X -13.7525,Y -79.3865,Z 81,A -104.2872,B 24.9187,C -2.0823,E1 24.9743,E2 188.9966} C_DIS
LIN {X -10.0371,Y -79.9405,Z 81,A -101.503,B 24.9185,C -2.085,E1 24.982,E2 186.2038} C_DIS
LIN {X -6.8562,Y -80.2765,Z 81,A -99.4901,B 24.9191,C -2.0772,E1 24.9876,E2 184.2084} C_DIS
LIN {X -3.9932,Y -80.4694,Z 81,A -96.7455,B 24.9175,C -2.098,E1 24.9954,E2 181.4135} C_DIS
LIN {X 0.5377,Y -80.5646,Z 81,A -94.9296,B 24.9206,C -2.0572,E1 25.0002,E2 179.6943} C_DIS
Enddeposition()
LIN {X 0.5377,Y -80.5646,Z 81,A -94.9296,B 24.9206,C -2.0572,E1 25.0002,E2 179.6943} C_DIS
Startdeposition()
$VEL.CP = VEL_PRINT
LIN {X -1.6359,Y -79.5643,Z 81,A -96.388,B 24.9191,C -2.0773,E1 24.9962,E2 181.1052} C_DIS
LIN {X -6.3476,Y -79.3274,Z 81,A -99.9411,B 24.9194,C -2.0726,E1 24.9863,E2 184.6704} C_DIS
LIN {X -9.865,Y -78.9671,Z 81,A -102.9247,B 24.9204,C -2.0606,E1 24.9779,E2 187.6844} C_DIS
LIN {X -13.0804,Y -78.4986,Z 81,A -105.541,B 24.9209,C -2.0536,E1 24.9707,E2 190.3199} C_DIS
LIN {X -16.4634,Y -77.8608,Z 81,A -107.7773,B 24.9203,C -2.0613,E1 24.9646,E2 192.5404} C_DIS
LIN {X -20.4399,Y -76.9119,Z 81,A -110.3387,B 24.9194,C -2.0735,E1 24.9577,E2 195.0765} C_DIS
LIN {X -23.2394,Y -76.1129,Z 81,A -112.5145,B 24.9194,C -2.0728,E1 24.9519,E2 197.2578} C_DIS
LIN {X -26.3535,Y -75.0907,Z 81,A -114.8037,B 24.9191,C -2.0766,E1 24.9458,E2 199.542} C_DIS
LIN {X -29.5662,Y -73.8863,Z 81,A -117.384,B 24.9191,C -2.0759,E1 24.9391,E2 202.1296} C_DIS
LIN {X -32.5392,Y -72.6248,Z 81,A -119.5814,B 24.9187,C -2.0819,E1 24.9335,E2 204.318} C_DIS
LIN {X -36.0643,Y -70.9402,Z 81,A -122.0326,B 24.9177,C -2.095,E1 24.9274,E2 206.7441} C_DIS
LIN {X -39.5724,Y -69.0446,Z 81,A -125.2626,B 24.9182,C -2.0891,E1 24.9194,E2 209.9975} C_DIS
LIN {X -43.5591,Y -66.6019,Z 81,A -128.3749,B 24.9172,C -2.1009,E1 24.9121,E2 213.0914} C_DIS
LIN {X -46.4982,Y -64.5845,Z 81,A -131.3359,B 24.9177,C -2.0946,E1 24.9052,E2 216.0777} C_DIS
LIN {X -50.079,Y -61.8484,Z 81,A -134.8087,B 24.9177,C -2.0944,E1 24.8976,E2 219.5637} C_DIS
LIN {X -53.2842,Y -59.11,Z 81,A -137.5113,B 24.9166,C -2.1089,E1 24.892,E2 222.2422} C_DIS
LIN {X -55.3558,Y -57.1742,Z 81,A -139.6311,B 24.9164,C -2.111,E1 24.8877,E2 224.3658} C_DIS
LIN {X -57.4183,Y -55.1026,Z 81,A -141.9149,B 24.9164,C -2.1108,E1 24.8832,E2 226.6599} C_DIS
LIN {X -60.0896,Y -52.1767,Z 81,A -144.7223,B 24.9158,C -2.1184,E1 24.878,E2 229.4619} C_DIS
LIN {X -62.6064,Y -49.1289,Z 81,A -147.2847,B 24.9147,C -2.1323,E1 24.8735,E2 232.003} C_DIS
LIN {X -64.2242,Y -46.9934,Z 81,A -149.9593,B 24.9159,C -2.1179,E1 24.869,E2 234.7248} C_DIS
LIN {X -66.4819,Y -43.7411,Z 81,A -152.2249,B 24.9141,C -2.14,E1 24.8655,E2 236.9491} C_DIS
LIN {X -68.1865,Y -41.0347,Z 81,A -154.6235,B 24.9138,C -2.1435,E1 24.862,E2 239.3515} C_DIS
LIN {X -70.3469,Y -37.2083,Z 81,A -157.733,B 24.913,C -2.1534,E1 24.8578,E2 242.4539} C_DIS
LIN {X -71.7842,Y -34.3536,Z 81,A -160.1583,B 24.9128,C -2.1566,E1 24.8548,E2 244.8846} C_DIS
LIN {X -73.3133,Y -30.9563,Z 81,A -163.1093,B 24.9128,C -2.1574,E1 24.8515,E2 247.85} C_DIS
LIN {X -74.5239,Y -27.9175,Z 81,A -165.2264,B 24.9117,C -2.1702,E1 24.8494,E2 249.9485} C_DIS
LIN {X -75.6115,Y -24.8222,Z 81,A -167.9452,B 24.9118,C -2.1682,E1 24.847,E2 252.6875} C_DIS
LIN {X -76.8832,Y -20.5463,Z 81,A -170.5144,B 24.9097,C -2.1939,E1 24.8451,E2 255.2101} C_DIS
LIN {X -77.4573,Y -18.2653,Z 81,A -172.5204,B 24.9099,C -2.1912,E1 24.8437,E2 257.2343} C_DIS
LIN {X -78.1528,Y -15.0087,Z 81,A -175.0442,B 24.9096,C -2.1955,E1 24.8423,E2 259.7629} C_DIS
LIN {X -78.7308,Y -11.6086,Z 81,A -177.4724,B 24.9088,C -2.2045,E1 24.8413,E2 262.1839} C_DIS
LIN {X -79.1536,Y -8.2367,Z 81,A -179.8082,B 24.908,C -2.215,E1 24.8405,E2 264.5087} C_DIS
LIN {X -79.4934,Y -3.7328,Z 81,A 176.7853,B 24.9074,C -2.2214,E1 24.8399,E2 267.9203} C_DIS
LIN {X -79.5804,Y 0.3624,Z 81,A 174.0171,B 24.9063,C -2.2353,E1 24.8398,E2 270.6721} C_DIS
LIN {X -79.5067,Y 3.4356,Z 81,A 171.342,B 24.9066,C -2.2309,E1 24.8401,E2 273.3738} C_DIS
LIN {X -79.2988,Y 6.7046,Z 81,A 168.802,B 24.9064,C -2.2339,E1 24.8406,E2 275.9219} C_DIS
LIN {X -78.8519,Y 10.756,Z 81,A 166.2615,B 24.9048,C -2.2529,E1 24.8415,E2 278.4321} C_DIS
LIN {X -78.3197,Y 14.1123,Z 81,A 163.8314,B 24.9041,C -2.2611,E1 24.8426,E2 280.8571} C_DIS
LIN {X -77.6584,Y 17.3925,Z 81,A 161.106,B 24.9041,C -2.2609,E1 24.8442,E2 283.5991} C_DIS
LIN {X -76.9119,Y 20.4399,Z 81,A 158.7416,B 24.9037,C -2.2653,E1 24.8459,E2 285.9666} C_DIS
LIN {X -75.8777,Y 23.9981,Z 81,A 156.3957,B 24.9023,C -2.2815,E1 24.8478,E2 288.2873} C_DIS
LIN {X -74.8025,Y 27.1612,Z 81,A 154.0746,B 24.9015,C -2.291,E1 24.85,E2 290.5989} C_DIS
LIN {X -73.6208,Y 30.2185,Z 81,A 151.6262,B 24.9011,C -2.296,E1 24.8525,E2 293.0492} C_DIS
LIN {X -71.375,Y 35.196,Z 81,A 147.8214,B 24.8998,C -2.3108,E1 24.8569,E2 296.8394} C_DIS
LIN {X -69.1897,Y 39.3187,Z 81,A 144.5476,B 24.8988,C -2.3227,E1 24.8613,E2 300.1021} C_DIS
LIN {X -67.3563,Y 42.383,Z 81,A 141.6981,B 24.8988,C -2.3229,E1 24.8654,E2 302.9658} C_DIS
LIN {X -65.5193,Y 45.1712,Z 81,A 138.84,B 24.8992,C -2.3181,E1 24.8699,E2 305.8494} C_DIS
LIN {X -62.5391,Y 49.2139,Z 81,A 135.2667,B 24.8982,C -2.3288,E1 24.876,E2 309.4143} C_DIS
LIN {X -60.2374,Y 52.0075,Z 81,A 133.0414,B 24.8968,C -2.345,E1 24.8799,E2 311.6111} C_DIS
LIN {X -58.1936,Y 54.2838,Z 81,A 130.8363,B 24.8963,C -2.3504,E1 24.8841,E2 313.813} C_DIS
LIN {X -55.2697,Y 57.2572,Z 81,A 127.5594,B 24.8963,C -2.3506,E1 24.8906,E2 317.1034} C_DIS
LIN {X -52.8556,Y 59.4937,Z 81,A 125.4322,B 24.8953,C -2.3622,E1 24.895,E2 319.2115} C_DIS
LIN {X -50.4284,Y 61.5652,Z 81,A 123.0906,B 24.895,C -2.3661,E1 24.9,E2 321.5528} C_DIS
LIN {X -47.1061,Y 64.1416,Z 81,A 119.5372,B 24.8956,C -2.3588,E1 24.908,E2 325.1362} C_DIS
LIN {X -44.4451,Y 66.0136,Z 81,A 118.3327,B 24.8925,C -2.3929,E1 24.9106,E2 326.2635} C_DIS
LIN {X -41.5043,Y 67.9011,Z 81,A 115.1958,B 24.8936,C -2.3814,E1 24.9181,E2 329.4379} C_DIS
LIN {X -39.0875,Y 69.321,Z 81,A 112.2923,B 24.8953,C -2.3619,E1 24.9253,E2 332.3963} C_DIS
LIN {X -35.3572,Y 71.2951,Z 81,A 110.1762,B 24.8927,C -2.3908,E1 24.9304,E2 334.4492} C_DIS
LIN {X -32.2452,Y 72.7562,Z 81,A 107.698,B 24.8924,C -2.3944,E1 24.9367,E2 336.9249} C_DIS
LIN {X -29.7383,Y 73.8162,Z 81,A 105.2116,B 24.8934,C -2.3832,E1 24.9432,E2 339.4434} C_DIS
LIN {X -25.7341,Y 75.306,Z 81,A 102.6046,B 24.892,C -2.3995,E1 24.95,E2 342.0168} C_DIS
LIN {X -22.7099,Y 76.2718,Z 81,A 100.3368,B 24.8917,C -2.4026,E1 24.956,E2 344.2813} C_DIS
LIN {X -18.699,Y 77.3531,Z 81,A 97.2538,B 24.8917,C -2.403,E1 24.9643,E2 347.3677} C_DIS
LIN {X -14.7482,Y 78.203,Z 81,A 94.1551,B 24.8919,C -2.4003,E1 24.9728,E2 350.4765} C_DIS
LIN {X -11.1711,Y 78.793,Z 81,A 91.1152,B 24.8928,C -2.3904,E1 24.9813,E2 353.5425} C_DIS
LIN {X -7.598,Y 79.2177,Z 81,A 89.2265,B 24.8909,C -2.4109,E1 24.9864,E2 355.3836} C_DIS
LIN {X -4.2623,Y 79.4667,Z 81,A 86.7398,B 24.891,C -2.4097,E1 24.9934,E2 357.874} C_DIS
LIN {X -1.0395,Y 79.5753,Z 81,A 84.2838,B 24.8913,C -2.4066,E1 25.0002,E2 360.3377} C_DIS
LIN {X 3.5061,Y 79.5037,Z 81,A 80.6224,B 24.8923,C -2.3961,E1 25.0105,E2 364.0229} C_DIS
LIN {X 6.7494,Y 79.294,Z 81,A 78.5115,B 24.8917,C -2.4024,E1 25.0164,E2 366.1179} C_DIS
LIN {X 10.9846,Y 78.8183,Z 81,A 75.5482,B 24.8915,C -2.4047,E1 25.0245,E2 369.0734} C_DIS
LIN {X 16.0376,Y 77.9482,Z 81,A 72.261,B 24.8906,C -2.4147,E1 25.0335,E2 372.3331} C_DIS
LIN {X 18.5298,Y 77.3944,Z 81,A 70.282,B 24.891,C -2.4097,E1 25.0389,E2 374.3212} C_DIS
LIN {X 21.3224,Y 76.6722,Z 81,A 68.1094,B 24.8914,C -2.4056,E1 25.0448,E2 376.5} C_DIS
LIN {X 24.6283,Y 75.6742,Z 81,A 65.6416,B 24.8915,C -2.4043,E1 25.0514,E2 378.9666} C_DIS
LIN {X 26.8762,Y 74.9064,Z 81,A 63.9807,B 24.8915,C -2.4042,E1 25.0557,E2 380.6243} C_DIS
LIN {X 29.7508,Y 73.8112,Z 81,A 61.8023,B 24.8916,C -2.4031,E1 25.0614,E2 382.8005} C_DIS
LIN {X 33.4265,Y 72.2206,Z 81,A 59.3246,B 24.8908,C -2.4118,E1 25.0677,E2 385.2515} C_DIS
LIN {X 36.9185,Y 70.4995,Z 81,A 56.2569,B 24.8919,C -2.4005,E1 25.0754,E2 388.3377} C_DIS
LIN {X 40.3992,Y 68.5642,Z 81,A 53.6344,B 24.8916,C -2.4038,E1 25.0817,E2 390.9447} C_DIS
LIN {X 42.3022,Y 67.4068,Z 81,A 51.6643,B 24.8928,C -2.3905,E1 25.0864,E2 392.9401} C_DIS
LIN {X 44.9015,Y 65.7046,Z 81,A 49.2996,B 24.8934,C -2.3831,E1 25.092,E2 395.3144} C_DIS
LIN {X 47.3351,Y 63.9738,Z 81,A 46.7032,B 24.8949,C -2.3661,E1 25.0979,E2 397.9417} C_DIS
LIN {X 49.9365,Y 61.9639,Z 81,A 45.242,B 24.8929,C -2.3889,E1 25.1009,E2 399.3436} C_DIS
LIN {X 51.6932,Y 60.5058,Z 81,A 43.2727,B 24.8941,C -2.3759,E1 25.1052,E2 401.3358} C_DIS
LIN {X 55.6413,Y 56.8975,Z 81,A 38.7059,B 24.8967,C -2.3466,E1 25.1146,E2 405.9532} C_DIS
LIN {X 58.3166,Y 54.1528,Z 81,A 35.9506,B 24.8972,C -2.3407,E1 25.1198,E2 408.7105} C_DIS
LIN {X 60.8561,Y 51.282,Z 81,A 33.9027,B 24.8959,C -2.3559,E1 25.1234,E2 410.7131} C_DIS
LIN {X 63.3796,Y 48.1282,Z 81,A 30.4619,B 24.8979,C -2.3327,E1 25.1294,E2 414.1924} C_DIS
LIN {X 65.346,Y 45.4205,Z 81,A 29.2078,B 24.8953,C -2.3622,E1 25.1313,E2 415.3708} C_DIS
LIN {X 67.3758,Y 42.3518,Z 81,A 26.0426,B 24.8973,C -2.3395,E1 25.1362,E2 418.574} C_DIS
LIN {X 69.109,Y 39.4604,Z 81,A 23.8124,B 24.8973,C -2.3391,E1 25.1393,E2 420.7934} C_DIS
LIN {X 70.8047,Y 36.3295,Z 81,A 21.2571,B 24.8979,C -2.3324,E1 25.1427,E2 423.3511} C_DIS
LIN {X 71.962,Y 33.9822,Z 81,A 18.8047,B 24.8999,C -2.3096,E1 25.1457,E2 425.8443} C_DIS
LIN {X 73.3667,Y 30.8296,Z 81,A 16.7032,B 24.8995,C -2.3144,E1 25.148,E2 427.923} C_DIS
LIN {X 74.5199,Y 27.9281,Z 81,A 14.4443,B 24.9001,C -2.3075,E1 25.1503,E2 430.1855} C_DIS
LIN {X 75.8125,Y 24.2009,Z 81,A 12.0241,B 24.8997,C -2.3123,E1 25.1524,E2 432.5807} C_DIS
LIN {X 76.8537,Y 20.6554,Z 81,A 8.3932,B 24.903,C -2.274,E1 25.1552,E2 436.2814} C_DIS
LIN {X 77.6938,Y 17.23,Z 81,A 6.668,B 24.9015,C -2.2917,E1 25.1562,E2 437.9548} C_DIS
LIN {X 78.1898,Y 14.8168,Z 81,A 4.1308,B 24.904,C -2.2623,E1 25.1576,E2 440.5466} C_DIS
LIN {X 78.7576,Y 11.4203,Z 81,A 2.3083,B 24.9029,C -2.2751,E1 25.1583,E2 442.3281} C_DIS
LIN {X 79.024,Y 9.3998,Z 81,A -0.0502,B 24.9057,C -2.2426,E1 25.1591,E2 444.7493} C_DIS
LIN {X 79.4117,Y 5.1909,Z 81,A -1.5386,B 24.9023,C -2.2819,E1 25.1594,E2 446.1361} C_DIS
LIN {X 79.5664,Y 1.5228,Z 81,A -5.2359,B 24.9059,C -2.2402,E1 25.1598,E2 449.91} C_DIS
LIN {X 79.4196,Y -5.0731,Z 81,A -9.1974,B 24.905,C -2.2499,E1 25.1594,E2 453.825} C_DIS
LIN {X 78.6699,Y -12.0084,Z 81,A -14.2465,B 24.9065,C -2.233,E1 25.1579,E2 458.884} C_DIS
LIN {X 77.5196,Y -17.9959,Z 81,A -18.7367,B 24.9079,C -2.2159,E1 25.1554,E2 463.3885} C_DIS
LIN {X 76.2723,Y -22.7082,Z 81,A -22.7567,B 24.9101,C -2.1889,E1 25.1524,E2 467.4492} C_DIS
LIN {X 74.7163,Y -27.3975,Z 81,A -25.8369,B 24.9098,C -2.1929,E1 25.1496,E2 470.5026} C_DIS
LIN {X 73.5524,Y -30.3865,Z 81,A -28.9837,B 24.9125,C -2.1597,E1 25.1462,E2 473.7105} C_DIS
LIN {X 71.9505,Y -34.0069,Z 81,A -30.8099,B 24.9106,C -2.1832,E1 25.1442,E2 475.4713} C_DIS
LIN {X 70.2451,Y -37.4016,Z 81,A -33.9694,B 24.9123,C -2.1618,E1 25.1401,E2 478.6645} C_DIS
LIN {X 67.9241,Y -41.4665,Z 81,A -37.2658,B 24.9129,C -2.1545,E1 25.1354,E2 481.9612} C_DIS
LIN {X 66.2587,Y -44.0797,Z 81,A -39.3416,B 24.913,C -2.1531,E1 25.1322,E2 484.0299} C_DIS
LIN {X 64.4268,Y -46.7166,Z 81,A -41.6394,B 24.9135,C -2.1472,E1 25.1285,E2 486.3304} C_DIS
LIN {X 62.0498,Y -49.8305,Z 81,A -44.4086,B 24.914,C -2.1414,E1 25.1238,E2 489.1004} C_DIS
LIN {X 60.4016,Y -51.8155,Z 81,A -46.209,B 24.9142,C -2.1383,E1 25.1205,E2 490.8998} C_DIS
LIN {X 58.4975,Y -53.9557,Z 81,A -48.2447,B 24.9146,C -2.134,E1 25.1167,E2 492.9367} C_DIS
LIN {X 56.3519,Y -56.1936,Z 81,A -50.6599,B 24.9155,C -2.1229,E1 25.1119,E2 495.3678} C_DIS
LIN {X 53.5836,Y -58.8389,Z 81,A -53.2339,B 24.9155,C -2.1221,E1 25.1067,E2 497.9332} C_DIS
LIN {X 51.3875,Y -60.7662,Z 81,A -55.2968,B 24.9158,C -2.1186,E1 25.1024,E2 499.9963} C_DIS
LIN {X 49.1718,Y -62.5724,Z 81,A -57.3566,B 24.9162,C -2.1141,E1 25.0979,E2 502.059} C_DIS
LIN {X 46.5587,Y -64.5413,Z 81,A -59.859,B 24.9169,C -2.1047,E1 25.0922,E2 504.5747} C_DIS
LIN {X 43.6716,Y -66.5277,Z 81,A -62.2755,B 24.9171,C -2.103,E1 25.0866,E2 506.9871} C_DIS
LIN {X 40.9566,Y -68.234,Z 81,A -64.6046,B 24.9175,C -2.098,E1 25.0811,E2 509.3206} C_DIS
LIN {X 38.1583,Y -69.8364,Z 81,A -66.9876,B 24.9179,C -2.0921,E1 25.0752,E2 511.7106} C_DIS
LIN {X 33.2065,Y -72.3231,Z 81,A -70.6272,B 24.9176,C -2.0962,E1 25.0662,E2 515.3307} C_DIS
LIN {X 31.0379,Y -73.2789,Z 81,A -72.984,B 24.9193,C -2.0743,E1 25.06,E2 517.7339} C_DIS
LIN {X 27.9209,Y -74.5227,Z 81,A -75.7669,B 24.9204,C -2.0602,E1 25.0527,E2 520.5441} C_DIS
LIN {X 24.1679,Y -75.8232,Z 81,A -77.6258,B 24.9184,C -2.0863,E1 25.0479,E2 522.3377} C_DIS
LIN {X 21.392,Y -76.6525,Z 81,A -79.9431,B 24.9191,C -2.0771,E1 25.0416,E2 524.6729} C_DIS
LIN {X 15.5801,Y -78.042,Z 81,A -83.874,B 24.9186,C -2.084,E1 25.031,E2 528.582} C_DIS
LIN {X 12.1281,Y -78.6513,Z 81,A -87.1956,B 24.9205,C -2.0589,E1 25.0217,E2 531.9598} C_DIS
LIN {X 8.4083,Y -79.1356,Z 81,A -90.6129,B 24.9222,C -2.0369,E1 25.0121,E2 535.4271} C_DIS
LIN {X 3.2726,Y -79.5137,Z 81,A -93.1443,B 24.9197,C -2.0689,E1 25.0052,E2 537.8816} C_DIS
LIN {X 0.5379,Y -79.5647,Z 81,A -94.9226,B 24.9193,C -2.0741,E1 25.0003,E2 539.6473} C_DIS
Enddeposition()
LIN {X 0.5379,Y -79.5647,Z 81,A -94.9226,B 24.9193,C -2.0741,E1 25.0003,E2 539.6473} C_DIS
Startdeposition()
$VEL.CP = VEL_PRINT
LIN {X 2.905,Y -78.5421,Z 81,A -92.3031,B 24.9159,C -2.1172,E1 25.0079,E2 536.9259} C_DIS
LIN {X 8.3215,Y -78.1527,Z 81,A -88.5457,B 24.9162,C -2.1133,E1 25.0183,E2 533.1798} C_DIS
LIN {X 14.4169,Y -77.2621,Z 81,A -83.9368,B 24.9157,C -2.1199,E1 25.0311,E2 528.5597} C_DIS
LIN {X 16.909,Y -76.754,Z 81,A -81.6475,B 24.9146,C -2.1344,E1 25.0374,E2 526.2388} C_DIS
LIN {X 21.6971,Y -75.5406,Z 81,A -78.4716,B 24.9153,C -2.1255,E1 25.0459,E2 523.0891} C_DIS
LIN {X 23.9367,Y -74.8611,Z 81,A -76.1725,B 24.9137,C -2.1453,E1 25.0521,E2 520.7474} C_DIS
LIN {X 26.9715,Y -73.8215,Z 81,A -74.5412,B 24.9151,C -2.1271,E1 25.0563,E2 519.1626} C_DIS
LIN {X 31.3811,Y -72.0576,Z 81,A -71.008,B 24.9146,C -2.1341,E1 25.0654,E2 515.6209} C_DIS
LIN {X 33.6782,Y -71.0138,Z 81,A -68.6289,B 24.913,C -2.1533,E1 25.0715,E2 513.2025} C_DIS
LIN {X 38.7085,Y -68.4026,Z 81,A -64.9437,B 24.9136,C -2.1468,E1 25.0805,E2 509.5433} C_DIS
LIN {X 41.4608,Y -66.7691,Z 81,A -62.7,B 24.9134,C -2.1484,E1 25.0859,E2 507.3029} C_DIS
LIN {X 43.5812,Y -65.4056,Z 81,A -60.4027,B 24.912,C -2.1661,E1 25.0913,E2 504.9714} C_DIS
LIN {X 47.9672,Y -62.2593,Z 81,A -57.019,B 24.9127,C -2.1572,E1 25.0988,E2 501.6206} C_DIS
LIN {X 50.4449,Y -60.2699,Z 81,A -54.6593,B 24.9122,C -2.1636,E1 25.1039,E2 499.2547} C_DIS
LIN {X 52.6206,Y -58.38,Z 81,A -52.3152,B 24.9112,C -2.176,E1 25.1089,E2 496.8908} C_DIS
LIN {X 56.059,Y -55.0863,Z 81,A -49.1177,B 24.9112,C -2.1758,E1 25.1152,E2 493.7072} C_DIS
LIN {X 58.2569,Y -52.758,Z 81,A -46.6884,B 24.9105,C -2.1845,E1 25.1198,E2 491.2679} C_DIS
LIN {X 59.9523,Y -50.8216,Z 81,A -44.6714,B 24.9097,C -2.1938,E1 25.1235,E2 489.2381} C_DIS
LIN {X 63.1546,Y -46.7841,Z 81,A -41.0957,B 24.9094,C -2.1981,E1 25.1296,E2 485.6692} C_DIS
LIN {X 65.0613,Y -44.092,Z 81,A -38.9153,B 24.9094,C -2.1976,E1 25.1331,E2 483.5006} C_DIS
LIN {X 67.4316,Y -40.3764,Z 81,A -35.6007,B 24.9084,C -2.2098,E1 25.138,E2 480.1739} C_DIS
LIN {X 69.8148,Y -36.0974,Z 81,A -32.0147,B 24.9075,C -2.2207,E1 25.1428,E2 476.581} C_DIS
LIN {X 71.5809,Y -32.4542,Z 81,A -28.8789,B 24.9063,C -2.2353,E1 25.1465,E2 473.4276} C_DIS
LIN {X 73.348,Y -28.2369,Z 81,A -25.762,B 24.906,C -2.2385,E1 25.1498,E2 470.3203} C_DIS
LIN {X 74.7583,Y -24.2542,Z 81,A -22.6325,B 24.9051,C -2.2496,E1 25.1526,E2 467.1822} C_DIS
LIN {X 76.188,Y -19.2994,Z 81,A -18.9782,B 24.9043,C -2.258,E1 25.1553,E2 463.5291} C_DIS
LIN {X 77.166,Y -14.9159,Z 81,A -15.3358,B 24.9025,C -2.2801,E1 25.1574,E2 459.8557} C_DIS
LIN {X 78.0462,Y -9.2673,Z 81,A -11.1306,B 24.9012,C -2.2946,E1 25.159,E2 455.6412} C_DIS
LIN {X 78.3907,Y -5.6664,Z 81,A -8.6543,B 24.9009,C -2.2978,E1 25.1595,E2 453.1719} C_DIS
LIN {X 78.585,Y -1.2291,Z 81,A -4.9038,B 24.8986,C -2.3246,E1 25.1598,E2 449.3806} C_DIS
LIN {X 78.5413,Y 2.9224,Z 81,A -2.7825,B 24.9003,C -2.3052,E1 25.1596,E2 447.3175} C_DIS
LIN {X 78.2683,Y 7.1505,Z 81,A 0.609,B 24.8986,C -2.3246,E1 25.1589,E2 443.9004} C_DIS
LIN {X 77.3448,Y 13.959,Z 81,A 5.3011,B 24.8981,C -2.3301,E1 25.1569,E2 439.2228} C_DIS
LIN {X 76.8372,Y 16.5279,Z 81,A 7.3379,B 24.8973,C -2.34,E1 25.1558,E2 437.1746} C_DIS
LIN {X 75.8753,Y 20.4941,Z 81,A 10.1382,B 24.8969,C -2.3436,E1 25.1538,E2 434.3821} C_DIS
LIN {X 74.9705,Y 23.5926,Z 81,A 12.9497,B 24.895,C -2.365,E1 25.1515,E2 431.536} C_DIS
LIN {X 73.4624,Y 27.935,Z 81,A 15.804,B 24.8956,C -2.3592,E1 25.1488,E2 428.7114} C_DIS
LIN {X 72.3627,Y 30.6715,Z 81,A 18.6749,B 24.893,C -2.388,E1 25.1456,E2 425.7882} C_DIS
LIN {X 70.825,Y 34.0719,Z 81,A 20.1643,B 24.8958,C -2.357,E1 25.144,E2 424.38} C_DIS
LIN {X 68.9042,Y 37.8078,Z 81,A 23.7256,B 24.8936,C -2.3808,E1 25.1393,E2 420.7813} C_DIS
LIN {X 66.8747,Y 41.2918,Z 81,A 26.6802,B 24.8929,C -2.389,E1 25.1351,E2 417.8225} C_DIS
LIN {X 65.0882,Y 44.0522,Z 81,A 28.6763,B 24.8935,C -2.3828,E1 25.132,E2 415.8511} C_DIS
LIN {X 63.2178,Y 46.6972,Z 81,A 31.4364,B 24.8918,C -2.4008,E1 25.1275,E2 413.0616} C_DIS
LIN {X 61.037,Y 49.5132,Z 81,A 33.9149,B 24.8916,C -2.4033,E1 25.1232,E2 410.5888} C_DIS
LIN {X 57.2418,Y 53.8558,Z 81,A 38.4072,B 24.89,C -2.4215,E1 25.1148,E2 406.0735} C_DIS
LIN {X 54.1008,Y 57.0114,Z 81,A 41.6828,B 24.8893,C -2.4291,E1 25.1082,E2 402.7935} C_DIS
LIN {X 50.7006,Y 60.0553,Z 81,A 44.6791,B 24.8896,C -2.4256,E1 25.102,E2 399.8175} C_DIS
LIN {X 47.0956,Y 62.9213,Z 81,A 48.3565,B 24.8882,C -2.4412,E1 25.0938,E2 396.1166} C_DIS
LIN {X 43.5043,Y 65.4563,Z 81,A 51.2185,B 24.8886,C -2.4361,E1 25.0872,E2 393.2762} C_DIS
LIN {X 40.7383,Y 67.2121,Z 81,A 54.4342,B 24.886,C -2.4645,E1 25.0794,E2 390.0035} C_DIS
LIN {X 37.1514,Y 69.2602,Z 81,A 56.4076,B 24.8885,C -2.4376,E1 25.0748,E2 388.0994} C_DIS
LIN {X 34.2489,Y 70.7399,Z 81,A 58.8698,B 24.888,C -2.4432,E1 25.0686,E2 385.6309} C_DIS
LIN {X 31.9141,Y 71.823,Z 81,A 61.0514,B 24.887,C -2.4543,E1 25.063,E2 383.4283} C_DIS
LIN {X 28.2355,Y 73.3486,Z 81,A 63.7739,B 24.8872,C -2.4518,E1 25.056,E2 380.7177} C_DIS
LIN {X 24.1512,Y 74.7917,Z 81,A 67.0596,B 24.8866,C -2.4582,E1 25.0473,E2 377.4234} C_DIS
LIN {X 20.6232,Y 75.8404,Z 81,A 69.475,B 24.8871,C -2.4523,E1 25.0408,E2 375.026} C_DIS
LIN {X 17.544,Y 76.6114,Z 81,A 71.6946,B 24.8873,C -2.4509,E1 25.0348,E2 372.8129} C_DIS
LIN {X 12.4958,Y 77.5961,Z 81,A 76.2523,B 24.885,C -2.4754,E1 25.0221,E2 368.2021} C_DIS
LIN {X 9.1199,Y 78.0634,Z 81,A 78.2896,B 24.8861,C -2.4631,E1 25.0166,E2 366.1955} C_DIS
LIN {X 4.4731,Y 78.4671,Z 81,A 81.5733,B 24.8864,C -2.4599,E1 25.0075,E2 362.9209} C_DIS
LIN {X -0.76,Y 78.5912,Z 81,A 85.5303,B 24.8861,C -2.4632,E1 24.9964,E2 358.9564} C_DIS
LIN {X -5.6787,Y 78.3898,Z 81,A 88.9388,B 24.8867,C -2.4569,E1 24.9869,E2 355.5621} C_DIS
LIN {X -8.7398,Y 78.1079,Z 81,A 91.207,B 24.8867,C -2.4565,E1 24.9806,E2 353.2935} C_DIS
LIN {X -12.6896,Y 77.5637,Z 81,A 94.1471,B 24.8868,C -2.4555,E1 24.9725,E2 350.3534} C_DIS
LIN {X -16.3143,Y 76.8833,Z 81,A 96.6972,B 24.8874,C -2.4495,E1 24.9655,E2 347.8145} C_DIS
LIN {X -18.9494,Y 76.2765,Z 81,A 99.2508,B 24.8861,C -2.4635,E1 24.9585,E2 345.2241} C_DIS
LIN {X -23.492,Y 75.0017,Z 81,A 102.1788,B 24.8877,C -2.4459,E1 24.9508,E2 342.3331} C_DIS
LIN {X -26.4283,Y 74.0189,Z 81,A 105.3547,B 24.8857,C -2.4679,E1 24.9423,E2 339.0986} C_DIS
LIN {X -30.3668,Y 72.4911,Z 81,A 107.099,B 24.8894,C -2.4278,E1 24.938,E2 337.4457} C_DIS
LIN {X -33.1242,Y 71.2732,Z 81,A 109.9922,B 24.888,C -2.443,E1 24.9305,E2 334.5094} C_DIS
LIN {X -37.0161,Y 69.3316,Z 81,A 112.9154,B 24.8891,C -2.4313,E1 24.9233,E2 331.6061} C_DIS
LIN {X -40.562,Y 67.3186,Z 81,A 116.3889,B 24.8883,C -2.4392,E1 24.9149,E2 328.1033} C_DIS
LIN {X -43.38,Y 65.5383,Z 81,A 119.3049,B 24.8876,C -2.4474,E1 24.9081,E2 325.1581} C_DIS
LIN {X -46.9881,Y 63.0021,Z 81,A 121.4565,B 24.8907,C -2.4129,E1 24.9034,E2 323.0812} C_DIS
LIN {X -49.9367,Y 60.6922,Z 81,A 124.3579,B 24.8909,C -2.4115,E1 24.897,E2 320.1724} C_DIS
LIN {X -52.2363,Y 58.724,Z 81,A 127.2558,B 24.8897,C -2.4244,E1 24.8909,E2 317.232} C_DIS
LIN {X -54.9556,Y 56.1882,Z 81,A 129.2858,B 24.8919,C -2.4004,E1 24.8869,E2 315.2508} C_DIS
LIN {X -57.8621,Y 53.1888,Z 81,A 132.2608,B 24.8927,C -2.3912,E1 24.8812,E2 312.2849} C_DIS
LIN {X -59.5907,Y 51.246,Z 81,A 135.1571,B 24.8908,C -2.4121,E1 24.8758,E2 309.3256} C_DIS
LIN {X -62.2838,Y 47.9354,Z 81,A 136.9692,B 24.8945,C -2.3707,E1 24.8729,E2 307.6036} C_DIS
LIN {X -64.0097,Y 45.6052,Z 81,A 139.8623,B 24.8933,C -2.3848,E1 24.868,E2 304.663} C_DIS
LIN {X -65.8934,Y 42.8409,Z 81,A 142.0117,B 24.8945,C -2.3707,E1 24.8648,E2 302.5364} C_DIS
LIN {X -67.7158,Y 39.8955,Z 81,A 144.8204,B 24.8945,C -2.3707,E1 24.8607,E2 299.7131} C_DIS
LIN {X -69.9004,Y 35.9311,Z 81,A 147.6572,B 24.8964,C -2.3495,E1 24.857,E2 296.912} C_DIS
LIN {X -71.5023,Y 32.6284,Z 81,A 150.5285,B 24.8967,C -2.3465,E1 24.8536,E2 294.0323} C_DIS
LIN {X -72.9566,Y 29.2333,Z 81,A 153.2471,B 24.8973,C -2.339,E1 24.8507,E2 291.3165} C_DIS
LIN {X -74.1272,Y 26.1198,Z 81,A 155.5812,B 24.8982,C -2.3293,E1 24.8484,E2 288.9923} C_DIS
LIN {X -75.1883,Y 22.8893,Z 81,A 158.5436,B 24.8978,C -2.3338,E1 24.8459,E2 286.0022} C_DIS
LIN {X -76.8079,Y 16.6621,Z 81,A 162.8176,B 24.9,C -2.3086,E1 24.8431,E2 281.7634} C_DIS
LIN {X -77.4392,Y 13.4338,Z 81,A 165.3058,B 24.9005,C -2.3033,E1 24.8419,E2 279.2732} C_DIS
LIN {X -77.844,Y 10.8367,Z 81,A 168.1663,B 24.8989,C -2.321,E1 24.8408,E2 276.3534} C_DIS
LIN {X -78.3255,Y 6.4992,Z 81,A 170.073,B 24.9026,C -2.2788,E1 24.8403,E2 274.5359} C_DIS
LIN {X -78.4683,Y 4.4516,Z 81,A 171.9401,B 24.9022,C -2.2833,E1 24.84,E2 272.6469} C_DIS
LIN {X -78.5843,Y 1.2664,Z 81,A 174.4229,B 24.9025,C -2.2798,E1 24.8398,E2 270.1573} C_DIS
LIN {X -78.5634,Y -2.2155,Z 81,A 177.0681,B 24.9029,C -2.2745,E1 24.8399,E2 267.5091} C_DIS
LIN {X -78.2932,Y -6.8818,Z 81,A -179.7921,B 24.9044,C -2.257,E1 24.8405,E2 264.3922} C_DIS
LIN {X -77.9709,Y -9.8819,Z 81,A -177.8328,B 24.9055,C -2.2441,E1 24.8412,E2 262.4519} C_DIS
LIN {X -77.5332,Y -12.8718,Z 81,A -174.9324,B 24.9046,C -2.2548,E1 24.8424,E2 259.5088} C_DIS
LIN {X -76.7311,Y -17.0144,Z 81,A -172.2439,B 24.9062,C -2.2355,E1 24.844,E2 256.8504} C_DIS
LIN {X -76.0906,Y -19.6801,Z 81,A -169.879,B 24.906,C -2.2387,E1 24.8456,E2 254.464} C_DIS
LIN {X -74.1977,Y -25.9187,Z 81,A -165.456,B 24.9079,C -2.2162,E1 24.8493,E2 250.0693} C_DIS
LIN {X -73.0807,Y -28.9181,Z 81,A -162.2574,B 24.9066,C -2.2316,E1 24.8526,E2 246.816} C_DIS
LIN {X -71.5231,Y -32.5826,Z 81,A -160.1823,B 24.909,C -2.2022,E1 24.8549,E2 244.7998} C_DIS
LIN {X -70.2221,Y -35.3006,Z 81,A -157.8165,B 24.9092,C -2.2005,E1 24.8579,E2 242.4254} C_DIS
LIN {X -67.3155,Y -40.5683,Z 81,A -153.5285,B 24.9103,C -2.1863,E1 24.8638,E2 238.1488} C_DIS
LIN {X -65.8863,Y -42.8519,Z 81,A -150.4508,B 24.9084,C -2.2102,E1 24.8686,E2 234.9985} C_DIS
LIN {X -63.1594,Y -46.7777,Z 81,A -148.0211,B 24.9113,C -2.1741,E1 24.8724,E2 232.6432} C_DIS
LIN {X -59.9022,Y -50.8803,Z 81,A -144.2923,B 24.9123,C -2.1629,E1 24.879,E2 228.9239} C_DIS
LIN {X -56.8078,Y -54.3143,Z 81,A -140.8336,B 24.9127,C -2.1578,E1 24.8855,E2 225.462} C_DIS
LIN {X -54.5862,Y -56.5458,Z 81,A -138.493,B 24.913,C -2.1542,E1 24.8902,E2 223.1201} C_DIS
LIN {X -52.1243,Y -58.8242,Z 81,A -136.2363,B 24.9138,C -2.1444,E1 24.8948,E2 220.8777} C_DIS
LIN {X -49.8348,Y -60.7754,Z 81,A -132.9263,B 24.9117,C -2.1702,E1 24.9021,E2 217.4937} C_DIS
LIN {X -46.4575,Y -63.3938,Z 81,A -130.7464,B 24.9141,C -2.1396,E1 24.9068,E2 215.3787} C_DIS
LIN {X -43.9562,Y -65.1532,Z 81,A -127.4469,B 24.9121,C -2.1651,E1 24.9146,E2 212.0076} C_DIS
LIN {X -40.0464,Y -67.6266,Z 81,A -125.1991,B 24.9149,C -2.1295,E1 24.9198,E2 209.8376} C_DIS
LIN {X -37.3002,Y -69.1795,Z 81,A -122.8478,B 24.9151,C -2.1278,E1 24.9256,E2 207.4836} C_DIS
LIN {X -34.2221,Y -70.7525,Z 81,A -120.2015,B 24.9151,C -2.1282,E1 24.9322,E2 204.8294} C_DIS
LIN {X -31.1013,Y -72.1796,Z 81,A -117.815,B 24.9155,C -2.1223,E1 24.9383,E2 202.4511} C_DIS
LIN {X -27.3233,Y -73.6932,Z 81,A -114.5815,B 24.9152,C -2.1269,E1 24.9467,E2 199.1999} C_DIS
LIN {X -23.9009,Y -74.8727,Z 81,A -112.1554,B 24.9158,C -2.1189,E1 24.9531,E2 196.7883} C_DIS
LIN {X -21.0274,Y -75.7304,Z 81,A -109.8687,B 24.9157,C -2.1203,E1 24.9593,E2 194.4947} C_DIS
LIN {X -15.7042,Y -77.0095,Z 81,A -105.8353,B 24.9157,C -2.1195,E1 24.9703,E2 190.4578} C_DIS
LIN {X -12.1653,Y -77.6473,Z 81,A -102.0265,B 24.9131,C -2.1528,E1 24.981,E2 186.5665} C_DIS
LIN {X -6.7438,Y -78.3059,Z 81,A -99.5673,B 24.9166,C -2.1086,E1 24.9876,E2 184.2109} C_DIS
LIN {X -1.9638,Y -78.5711,Z 81,A -96.0967,B 24.9166,C -2.1083,E1 24.9973,E2 180.7401} C_DIS
LIN {X 0.529,Y -78.5633,Z 81,A -94.4715,B 24.917,C -2.1037,E1 25.0018,E2 179.1259} C_DIS
Enddeposition()
LIN {X 0.529,Y -78.5633,Z 81,A -94.4715,B 24.917,C -2.1037,E1 25.0018,E2 179.1259} C_DIS
Startdeposition()
$VEL.CP = VEL_PRINT
LIN {X -0.9077,Y -77.6033,Z 81,A -96.1748,B 24.9171,C -2.102,E1 24.997,E2 180.8332} C_DIS
LIN {X -4.7533,Y -77.4635,Z 81,A -98.9491,B 24.9171,C -2.1036,E1 24.9892,E2 183.6044} C_DIS
LIN {X -7.5223,Y -77.2433,Z 81,A -102.1133,B 24.9194,C -2.0734,E1 24.9803,E2 186.8421} C_DIS
LIN {X -11.8958,Y -76.6907,Z 81,A -104.74,B 24.918,C -2.0911,E1 24.9731,E2 189.4288} C_DIS
LIN {X -15.0533,Y -76.1348,Z 81,A -107.8299,B 24.9194,C -2.0727,E1 24.9645,E2 192.5662} C_DIS
LIN {X -19.6277,Y -75.0854,Z 81,A -110.2505,B 24.9171,C -2.1025,E1 24.9581,E2 194.9193} C_DIS
LIN {X -22.7009,Y -74.214,Z 81,A -112.5841,B 24.9169,C -2.1047,E1 24.9519,E2 197.2514} C_DIS
LIN {X -26.7918,Y -72.8369,Z 81,A -116.473,B 24.9182,C -2.0888,E1 24.9415,E2 201.1858} C_DIS
LIN {X -30.132,Y -71.5194,Z 81,A -118.1366,B 24.9159,C -2.1176,E1 24.9374,E2 202.7848} C_DIS
LIN {X -32.3198,Y -70.5586,Z 81,A -120.9352,B 24.9179,C -2.0923,E1 24.9301,E2 205.6503} C_DIS
LIN {X -35.6592,Y -68.9314,Z 81,A -123.3537,B 24.917,C -2.1042,E1 24.9242,E2 208.0472} C_DIS
LIN {X -39.1303,Y -67.0221,Z 81,A -126.4636,B 24.917,C -2.1034,E1 24.9166,E2 211.1681} C_DIS
LIN {X -41.8649,Y -65.3475,Z 81,A -128.7492,B 24.9166,C -2.1091,E1 24.9113,E2 213.4474} C_DIS
LIN {X -44.8779,Y -63.3167,Z 81,A -131.5252,B 24.9164,C -2.1111,E1 24.9049,E2 216.2282} C_DIS
LIN {X -47.4711,Y -61.3961,Z 81,A -133.7364,B 24.9157,C -2.1197,E1 24.9,E2 218.427} C_DIS
LIN {X -50.7742,Y -58.6948,Z 81,A -136.5234,B 24.9145,C -2.1349,E1 24.8941,E2 221.1887} C_DIS
LIN {X -53.2807,Y -56.4283,Z 81,A -139.074,B 24.9142,C -2.1384,E1 24.8889,E2 223.7411} C_DIS
LIN {X -54.9867,Y -54.768,Z 81,A -140.7901,B 24.9139,C -2.1431,E1 24.8855,E2 225.4533} C_DIS
LIN {X -58.5681,Y -50.9193,Z 81,A -144.4459,B 24.9127,C -2.1573,E1 24.8787,E2 229.0913} C_DIS
LIN {X -61.2081,Y -47.715,Z 81,A -147.7047,B 24.9125,C -2.1596,E1 24.8729,E2 232.3599} C_DIS
LIN {X -63.9206,Y -44.014,Z 81,A -151.6863,B 24.913,C -2.1532,E1 24.8664,E2 236.3762} C_DIS
LIN {X -67.1845,Y -38.849,Z 81,A -155.9497,B 24.9116,C -2.1711,E1 24.8602,E2 240.6189} C_DIS
LIN {X -69.4957,Y -34.5444,Z 81,A -159.014,B 24.9097,C -2.1942,E1 24.8563,E2 243.6442} C_DIS
LIN {X -70.5312,Y -32.3803,Z 81,A -161.565,B 24.9109,C -2.18,E1 24.8533,E2 246.243} C_DIS
LIN {X -72.7654,Y -26.9879,Z 81,A -165.9724,B 24.91,C -2.1901,E1 24.8488,E2 250.651} C_DIS
LIN {X -74.3968,Y -22.0926,Z 81,A -169.2789,B 24.9081,C -2.2136,E1 24.846,E2 253.9204} C_DIS
LIN {X -75.2949,Y -18.8104,Z 81,A -171.6177,B 24.9071,C -2.2254,E1 24.8443,E2 256.2447} C_DIS
LIN {X -75.8852,Y -16.2629,Z 81,A -173.9901,B 24.9075,C -2.2206,E1 24.8429,E2 258.6425} C_DIS
LIN {X -76.5633,Y -12.6901,Z 81,A -176.313,B 24.9061,C -2.2376,E1 24.8418,E2 260.9384} C_DIS
LIN {X -76.9905,Y -9.7706,Z 81,A -178.4044,B 24.9053,C -2.2465,E1 24.841,E2 263.0211} C_DIS
LIN {X -77.2537,Y -7.41,Z 81,A 179.3807,B 24.9058,C -2.2409,E1 24.8403,E2 265.2628} C_DIS
LIN {X -77.5824,Y -2.0176,Z 81,A 175.6176,B 24.9043,C -2.2589,E1 24.8398,E2 269.0054} C_DIS
LIN {X -77.6021,Y 1.0205,Z 81,A 172.2867,B 24.9059,C -2.2402,E1 24.8399,E2 272.4012} C_DIS
LIN {X -77.4152,Y 5.4689,Z 81,A 170.2648,B 24.9024,C -2.2808,E1 24.8403,E2 274.3383} C_DIS
LIN {X -76.8704,Y 10.6755,Z 81,A 166.1667,B 24.9018,C -2.2874,E1 24.8415,E2 278.445} C_DIS
LIN {X -76.5236,Y 12.9273,Z 81,A 164.4168,B 24.9015,C -2.2911,E1 24.8423,E2 280.1964} C_DIS
LIN {X -75.9234,Y 16.0879,Z 81,A 161.0393,B 24.9029,C -2.2748,E1 24.8443,E2 283.633} C_DIS
LIN {X -74.9129,Y 20.2735,Z 81,A 158.7505,B 24.9002,C -2.3059,E1 24.8458,E2 285.8608} C_DIS
LIN {X -73.7825,Y 24.0654,Z 81,A 155.6267,B 24.8999,C -2.3101,E1 24.8484,E2 288.9926} C_DIS
LIN {X -72.709,Y 27.1386,Z 81,A 153.134,B 24.8994,C -2.3152,E1 24.8508,E2 291.487} C_DIS
LIN {X -71.2399,Y 30.788,Z 81,A 150.4025,B 24.8983,C -2.3281,E1 24.8538,E2 294.2029} C_DIS
LIN {X -69.4668,Y 34.6027,Z 81,A 147.5473,B 24.897,C -2.3434,E1 24.8572,E2 297.0372} C_DIS
LIN {X -67.0501,Y 39.0811,Z 81,A 143.2585,B 24.8971,C -2.3413,E1 24.863,E2 301.3535} C_DIS
LIN {X -65.2685,Y 41.9881,Z 81,A 141.0777,B 24.8958,C -2.3565,E1 24.8662,E2 303.5091} C_DIS
LIN {X -61.904,Y 46.8073,Z 81,A 137.0302,B 24.8941,C -2.3754,E1 24.8727,E2 307.5314} C_DIS
LIN {X -58.8666,Y 50.5746,Z 81,A 133.3838,B 24.8935,C -2.3828,E1 24.8792,E2 311.177} C_DIS
LIN {X -56.6213,Y 53.0755,Z 81,A 130.3458,B 24.8941,C -2.3752,E1 24.8849,E2 314.2465} C_DIS
LIN {X -54.6398,Y 55.1134,Z 81,A 127.3293,B 24.8957,C -2.3578,E1 24.8911,E2 317.3172} C_DIS
LIN {X -50.9976,Y 58.4997,Z 81,A 125.4232,B 24.891,C -2.4097,E1 24.8948,E2 319.1072} C_DIS
LIN {X -48.5261,Y 60.566,Z 81,A 122.2421,B 24.8924,C -2.3947,E1 24.9017,E2 322.336} C_DIS
LIN {X -43.6335,Y 64.1803,Z 81,A 118.1997,B 24.8905,C -2.4151,E1 24.9108,E2 326.3441} C_DIS
LIN {X -41.5949,Y 65.5209,Z 81,A 115.093,B 24.8932,C -2.3857,E1 24.9183,E2 329.5306} C_DIS
LIN {X -37.7503,Y 67.8077,Z 81,A 112.3631,B 24.8914,C -2.4058,E1 24.9248,E2 332.2207} C_DIS
LIN {X -34.8744,Y 69.3322,Z 81,A 109.922,B 24.8911,C -2.4086,E1 24.9309,E2 334.6615} C_DIS
LIN {X -30.4832,Y 71.3714,Z 81,A 106.5503,B 24.8902,C -2.4191,E1 24.9395,E2 338.0166} C_DIS
LIN {X -26.3239,Y 73.0075,Z 81,A 103.7532,B 24.8886,C -2.4364,E1 24.9467,E2 340.7783} C_DIS
LIN {X -24.195,Y 73.7405,Z 81,A 101.3204,B 24.8902,C -2.4184,E1 24.9533,E2 343.2585} C_DIS
LIN {X -20.2509,Y 74.9191,Z 81,A 98.9506,B 24.8884,C -2.439,E1 24.9595,E2 345.5829} C_DIS
LIN {X -17.4055,Y 75.6308,Z 81,A 96.5282,B 24.8888,C -2.4343,E1 24.9661,E2 348.0199} C_DIS
LIN {X -14.303,Y 76.2793,Z 81,A 94.2896,B 24.8884,C -2.4388,E1 24.9722,E2 350.2502} C_DIS
LIN {X -9.9078,Y 76.9727,Z 81,A 90.7936,B 24.8887,C -2.4354,E1 24.9819,E2 353.7572} C_DIS
LIN {X -6.9919,Y 77.2923,Z 81,A 88.7506,B 24.8883,C -2.4398,E1 24.9876,E2 355.791} C_DIS
LIN {X -1.6061,Y 77.5911,Z 81,A 84.9724,B 24.8877,C -2.4466,E1 24.9981,E2 359.5538} C_DIS
LIN {X 1.1876,Y 77.599,Z 81,A 82.7636,B 24.888,C -2.443,E1 25.0042,E2 361.771} C_DIS
LIN {X 5.2231,Y 77.4318,Z 81,A 79.6701,B 24.8883,C -2.4401,E1 25.0129,E2 364.8704} C_DIS
LIN {X 8.9001,Y 77.0958,Z 81,A 76.7294,B 24.8888,C -2.4339,E1 25.0211,E2 367.8239} C_DIS
LIN {X 11.757,Y 76.7121,Z 81,A 73.7249,B 24.8911,C -2.4094,E1 25.0296,E2 370.8835} C_DIS
LIN {X 16.693,Y 75.7914,Z 81,A 71.3397,B 24.8879,C -2.4439,E1 25.0358,E2 373.1839} C_DIS
LIN {X 19.4938,Y 75.1198,Z 81,A 69.0836,B 24.8883,C -2.4391,E1 25.042,E2 375.4482} C_DIS
LIN {X 23.6741,Y 73.9091,Z 81,A 65.2219,B 24.8902,C -2.4186,E1 25.0524,E2 379.3513} C_DIS
LIN {X 27.0051,Y 72.7591,Z 81,A 63.2699,B 24.8888,C -2.4344,E1 25.0574,E2 381.2618} C_DIS
LIN {X 29.8989,Y 71.6176,Z 81,A 60.5234,B 24.8901,C -2.4194,E1 25.0646,E2 384.0376} C_DIS
LIN {X 32.9708,Y 70.2563,Z 81,A 58.1386,B 24.8901,C -2.4192,E1 25.0706,E2 386.4168} C_DIS
LIN {X 36.2856,Y 68.6028,Z 81,A 55.3704,B 24.8906,C -2.4148,E1 25.0774,E2 389.1879} C_DIS
LIN {X 41.0818,Y 65.8427,Z 81,A 51.8835,B 24.8895,C -2.426,E1 25.0857,E2 392.6374} C_DIS
LIN {X 43.4544,Y 64.3015,Z 81,A 48.7426,B 24.8926,C -2.3924,E1 25.0932,E2 395.8473} C_DIS
LIN {X 46.8558,Y 61.8674,Z 81,A 46.38,B 24.8912,C -2.4079,E1 25.0984,E2 398.1648} C_DIS
LIN {X 49.8808,Y 59.4559,Z 81,A 43.5201,B 24.8917,C -2.4025,E1 25.1045,E2 401.0267} C_DIS
LIN {X 52.4617,Y 57.1903,Z 81,A 41.2923,B 24.8913,C -2.4065,E1 25.1091,E2 403.2361} C_DIS
LIN {X 54.6702,Y 55.0832,Z 81,A 38.9076,B 24.8921,C -2.3979,E1 25.1139,E2 405.631} C_DIS
LIN {X 59.3086,Y 50.0558,Z 81,A 34.15,B 24.8923,C -2.3954,E1 25.1228,E2 410.3736} C_DIS
LIN {X 61.0195,Y 47.9544,Z 81,A 31.3077,B 24.895,C -2.3657,E1 25.1279,E2 413.2728} C_DIS
LIN {X 63.0538,Y 45.2462,Z 81,A 29.445,B 24.8938,C -2.3785,E1 25.1308,E2 415.0962} C_DIS
LIN {X 64.5588,Y 43.0732,Z 81,A 27.4513,B 24.8944,C -2.3723,E1 25.134,E2 417.0947} C_DIS
LIN {X 67.1377,Y 38.9305,Z 81,A 24.2551,B 24.8941,C -2.3752,E1 25.1386,E2 420.2679} C_DIS
LIN {X 68.2297,Y 36.9822,Z 81,A 21.6816,B 24.897,C -2.3429,E1 25.1421,E2 422.9041} C_DIS
LIN {X 69.7727,Y 33.9839,Z 81,A 19.8102,B 24.896,C -2.3546,E1 25.1444,E2 424.7379} C_DIS
LIN {X 71.6275,Y 29.8755,Z 81,A 16.5099,B 24.8967,C -2.346,E1 25.1481,E2 428.0405} C_DIS
Enddeposition()
END
